LIN {X 0,Y 252.438,Z 584.702,A -85,B 0,C 180,E1 -18965.317,E2 -18965.317} C_VEL
LIN {X 0,Y 250.737,Z 589.425,A -85,B 0,C 180,E1 -18967.666,E2 -18967.666} C_VEL
LIN {X 0,Y 249.329,Z 593.32,A -85,B 0,C 180,E1 -18970.23,E2 -18970.23} C_VEL
LIN {X 0,Y 248.647,Z 595.228,A -85,B 0,C 180,E1 -18971.886,E2 -18971.886} C_VEL
LIN {X 0,Y 247.812,Z 597.412,A -85,B 0,C 180,E1 -18974.635,E2 -18974.635} C_VEL
LIN {X 0,Y 247.334,Z 598.311,A -85,B 0,C 180,E1 -18976.861,E2 -18976.861} C_VEL
LIN {X 0,Y 247.03,Z 598.544,A -85,B 0,C 180,E1 -18978.513,E2 -18978.513} C_VEL
LIN {X 0,Y 246.93,Z 598.348,A -85,B 0,C 180,E1 -18980.168,E2 -18980.168} C_VEL
LIN {X 0,Y 246.961,Z 597.738,A -85,B 0,C 180,E1 -18981.82,E2 -18981.82} C_VEL
LIN {X 0,Y 247.195,Z 596.06,A -85,B 0,C 180,E1 -18984.324,E2 -18984.324} C_VEL
LIN {X 0,Y 247.49,Z 592.461,A -85,B 0,C 180,E1 -18987.559,E2 -18987.559} C_VEL
LIN {X 0,Y 248.083,Z 588.535,A -85,B 0,C 180,E1 -18990,E2 -18990} C_VEL
LIN {X 0,Y 248.817,Z 583.495,A -85,B 0,C 180,E1 -18992.428,E2 -18992.428} C_VEL
LIN {X 0,Y 249.968,Z 577.141,A -85,B 0,C 180,E1 -18994.838,E2 -18994.838} C_VEL
LIN {X 0,Y 251.454,Z 569.206,A -85,B 0,C 180,E1 -18997.225,E2 -18997.225} C_VEL
LIN {X 0,Y 253.19,Z 559.359,A -85,B 0,C 180,E1 -18999.587,E2 -18999.587} C_VEL
LIN {X 0,Y 254.996,Z 549.004,A -85,B 0,C 180,E1 -19001.526,E2 -19001.526} C_VEL
LIN {X 0,Y 256.526,Z 538.775,A -85,B 0,C 180,E1 -19003.063,E2 -19003.063} C_VEL
LIN {X 0,Y 257.87,Z 527.613,A -85,B 0,C 180,E1 -19004.4,E2 -19004.4} C_VEL
LIN {X 0,Y 259.068,Z 516.263,A -85,B 0,C 180,E1 -19005.438,E2 -19005.438} C_VEL
LIN {X 0,Y 260.042,Z 503.315,A -85,B 0,C 180,E1 -19006.284,E2 -19006.284} C_VEL
LIN {X 0,Y 260.587,Z 491.019,A -85,B 0,C 180,E1 -19006.803,E2 -19006.803} C_VEL
LIN {X 0,Y 262.544,Z 423.316,A -85,B 0,C 180,E1 -19008.621,E2 -19008.621} C_VEL
LIN {X 0,Y 256.099,Z 405.689,A -85,B 0,C 180,E1 -19009.811,E2 -19009.811} C_VEL
LIN {X 0,Y 249.864,Z 392.807,A -85,B 0,C 180,E1 -19010.9,E2 -19010.9} C_VEL
LIN {X 0,Y 249.121,Z 390.454,A -85,B 0,C 180,E1 -19011.108,E2 -19011.108} C_VEL
LIN {X 0,Y 249.136,Z 390.441,A -85,B 0,C 180,E1 -19015.482,E2 -19015.482} C_VEL
LIN {X 0,Y 249.09,Z 390.455,A -85,B 0,C 180,E1 -19018.994,E2 -19018.994} C_VEL
LIN {X 0,Y 249.035,Z 390.465,A -85,B 0,C 180,E1 -19022.424,E2 -19022.424} C_VEL
LIN {X 0,Y 249.059,Z 390.462,A -85,B 0,C 180,E1 -19026.339,E2 -19026.339} C_VEL
LIN {X 0,Y 249.008,Z 390.46,A -85,B 0,C 180,E1 -19030.477,E2 -19030.477} C_VEL
LIN {X 0,Y 249.018,Z 390.463,A -85,B 0,C 180,E1 -19034.874,E2 -19034.874} C_VEL
LIN {X 0,Y 249.08,Z 390.445,A -85,B 0,C 180,E1 -19037.376,E2 -19037.376} C_VEL
LIN {X 0,Y 249.052,Z 390.46,A -85,B 0,C 180,E1 -19041.623,E2 -19041.623} C_VEL
LIN {X 0,Y 249.059,Z 390.445,A -85,B 0,C 180,E1 -19045.641,E2 -19045.641} C_VEL
LIN {X 0,Y 249.045,Z 390.461,A -85,B 0,C 180,E1 -19049.471,E2 -19049.471} C_VEL
LIN {X 0,Y 249.068,Z 390.449,A -85,B 0,C 180,E1 -19053.161,E2 -19053.161} C_VEL
LIN {X 0,Y 249.081,Z 390.455,A -85,B 0,C 180,E1 -19056.732,E2 -19056.732} C_VEL
LIN {X 0,Y 249.127,Z 390.453,A -85,B 0,C 180,E1 -19060.212,E2 -19060.212} C_VEL
LIN {X 0,Y 249.238,Z 390.426,A -85,B 0,C 180,E1 -19063.621,E2 -19063.621} C_VEL
LIN {X 0,Y 249.248,Z 390.436,A -85,B 0,C 180,E1 -19068.616,E2 -19068.616} C_VEL
LIN {X 0,Y 249.476,Z 390.406,A -85,B 0,C 180,E1 -19071.902,E2 -19071.902} C_VEL
LIN {X 0,Y 249.431,Z 390.406,A -85,B 0,C 180,E1 -19076.769,E2 -19076.769} C_VEL
LIN {X 0,Y 249.73,Z 390.378,A -85,B 0,C 180,E1 -19080,E2 -19080} C_VEL
LIN {X 0,Y 249.432,Z 390.408,A -85,B 0,C 180,E1 -19083.23,E2 -19083.23} C_VEL
LIN {X 0,Y 249.476,Z 390.407,A -85,B 0,C 180,E1 -19088.097,E2 -19088.097} C_VEL
LIN {X 0,Y 249.354,Z 390.421,A -85,B 0,C 180,E1 -19089.954,E2 -19089.954} C_VEL
LIN {X 0,Y 248.581,Z 390.52,A -85,B 0,C 180,E1 -19091.3,E2 -19091.3} C_VEL
LIN {X 0,Y 245.714,Z 390.878,A -85,B 0,C 180,E1 -19093.495,E2 -19093.495} C_VEL
LIN {X 0,Y 242.486,Z 391.281,A -85,B 0,C 180,E1 -19096.2,E2 -19096.2} C_VEL
LIN {X 0,Y 242.121,Z 391.321,A -85,B 0,C 180,E1 -19097.136,E2 -19097.136} C_VEL
LIN {X 0,Y 242.045,Z 391.335,A -85,B 0,C 180,E1 -19102.177,E2 -19102.177} C_VEL
LIN {X 0,Y 242.062,Z 391.335,A -85,B 0,C 180,E1 -19105.838,E2 -19105.838} C_VEL
LIN {X 0,Y 242.003,Z 391.34,A -85,B 0,C 180,E1 -19109.584,E2 -19109.584} C_VEL
LIN {X 0,Y 241.987,Z 391.343,A -85,B 0,C 180,E1 -19113.491,E2 -19113.491} C_VEL
LIN {X 0,Y 242.009,Z 391.34,A -85,B 0,C 180,E1 -19117.578,E2 -19117.578} C_VEL
LIN {X 0,Y 241.982,Z 391.342,A -85,B 0,C 180,E1 -19121.913,E2 -19121.913} C_VEL
LIN {X 0,Y 241.97,Z 391.344,A -85,B 0,C 180,E1 -19126.562,E2 -19126.562} C_VEL
LIN {X 0,Y 241.976,Z 391.346,A -85,B 0,C 180,E1 -19130.286,E2 -19130.286} C_VEL
LIN {X 0,Y 242.073,Z 391.536,A -85,B 0,C 180,E1 -19132.906,E2 -19132.906} C_VEL
LIN {X 0,Y 244.318,Z 401.427,A -85,B 0,C 180,E1 -19136.87,E2 -19136.87} C_VEL
LIN {X 0,Y 245.764,Z 408.526,A -85,B 0,C 180,E1 -19139.488,E2 -19139.488} C_VEL
LIN {X 0,Y 250.251,Z 420.691,A -85,B 0,C 180,E1 -19140.38,E2 -19140.38} C_VEL
LIN {X 0,Y 254.146,Z 451.891,A -85,B 0,C 180,E1 -19141.755,E2 -19141.755} C_VEL
LIN {X 0,Y 255.201,Z 463.108,A -85,B 0,C 180,E1 -19142.202,E2 -19142.202} C_VEL
LIN {X 0,Y 253.446,Z 517.374,A -85,B 0,C 180,E1 -19143.717,E2 -19143.717} C_VEL
LIN {X 0,Y 252.497,Z 530.59,A -85,B 0,C 180,E1 -19144.387,E2 -19144.387} C_VEL
LIN {X 0,Y 251.165,Z 542.728,A -85,B 0,C 180,E1 -19145.294,E2 -19145.294} C_VEL
LIN {X 0,Y 249.537,Z 554.986,A -85,B 0,C 180,E1 -19146.559,E2 -19146.559} C_VEL
LIN {X 0,Y 247.702,Z 566.611,A -85,B 0,C 180,E1 -19148.137,E2 -19148.137} C_VEL
LIN {X 0,Y 245.775,Z 577.065,A -85,B 0,C 180,E1 -19149.932,E2 -19149.932} C_VEL
LIN {X 0,Y 244.06,Z 587.411,A -85,B 0,C 180,E1 -19152.213,E2 -19152.213} C_VEL
LIN {X 0,Y 242.628,Z 595.579,A -85,B 0,C 180,E1 -19154.459,E2 -19154.459} C_VEL
LIN {X 0,Y 241.355,Z 602.896,A -85,B 0,C 180,E1 -19156.958,E2 -19156.958} C_VEL
LIN {X 0,Y 240.678,Z 607.838,A -85,B 0,C 180,E1 -19159.059,E2 -19159.059} C_VEL
LIN {X 0,Y 240.168,Z 612.631,A -85,B 0,C 180,E1 -19161.587,E2 -19161.587} C_VEL
LIN {X 0,Y 239.979,Z 615.204,A -85,B 0,C 180,E1 -19163.273,E2 -19163.273} C_VEL
LIN {X 0,Y 239.92,Z 617.267,A -85,B 0,C 180,E1 -19164.958,E2 -19164.958} C_VEL
LIN {X 0,Y 239.952,Z 618.906,A -85,B 0,C 180,E1 -19166.642,E2 -19166.642} C_VEL
LIN {X 0,Y 240.006,Z 620.132,A -85,B 0,C 180,E1 -19168.322,E2 -19168.322} C_VEL
LIN {X 0,Y 240.02,Z 620.919,A -85,B 0,C 180,E1 -19170,E2 -19170} C_VEL
LIN {X 0,Y 239.975,Z 621.281,A -85,B 0,C 180,E1 -19171.678,E2 -19171.678} C_VEL
LIN {X 0,Y 239.902,Z 621.251,A -85,B 0,C 180,E1 -19173.359,E2 -19173.359} C_VEL
LIN {X 0,Y 239.845,Z 620.834,A -85,B 0,C 180,E1 -19175.043,E2 -19175.043} C_VEL
LIN {X 0,Y 239.9,Z 620.017,A -85,B 0,C 180,E1 -19176.729,E2 -19176.729} C_VEL
LIN {X 0,Y 240.552,Z 617.129,A -85,B 0,C 180,E1 -19180.096,E2 -19180.096} C_VEL
LIN {X 0,Y 241.429,Z 613.857,A -85,B 0,C 180,E1 -19182.61,E2 -19182.61} C_VEL
LIN {X 0,Y 242.806,Z 609.541,A -85,B 0,C 180,E1 -19185.1,E2 -19185.1} C_VEL
LIN {X 0,Y 244.64,Z 604.063,A -85,B 0,C 180,E1 -19187.556,E2 -19187.556} C_VEL
LIN {X 0,Y 246.842,Z 597.119,A -85,B 0,C 180,E1 -19190.021,E2 -19190.021} C_VEL
LIN {X 0,Y 249.439,Z 588.791,A -85,B 0,C 180,E1 -19192.356,E2 -19192.356} C_VEL
LIN {X 0,Y 252.13,Z 580.114,A -85,B 0,C 180,E1 -19194.276,E2 -19194.276} C_VEL
LIN {X 0,Y 255.107,Z 569.459,A -85,B 0,C 180,E1 -19196.153,E2 -19196.153} C_VEL
LIN {X 0,Y 257.715,Z 558.887,A -85,B 0,C 180,E1 -19197.619,E2 -19197.619} C_VEL
LIN {X 0,Y 260.14,Z 547.118,A -85,B 0,C 180,E1 -19198.875,E2 -19198.875} C_VEL
LIN {X 0,Y 262.356,Z 533.614,A -85,B 0,C 180,E1 -19199.928,E2 -19199.928} C_VEL
LIN {X 0,Y 263.864,Z 520.48,A -85,B 0,C 180,E1 -19200.622,E2 -19200.622} C_VEL
LIN {X 0,Y 264.804,Z 504.801,A -85,B 0,C 180,E1 -19201.107,E2 -19201.107} C_VEL
LIN {X 0,Y 266.35,Z 464.818,A -85,B 0,C 180,E1 -19202.171,E2 -19202.171} C_VEL
LIN {X 0,Y 262.808,Z 441.78,A -85,B 0,C 180,E1 -19203.496,E2 -19203.496} C_VEL
LIN {X 0,Y 261.785,Z 438.425,A -85,B 0,C 180,E1 -19203.778,E2 -19203.778} C_VEL
LIN {X 0,Y 254.825,Z 423.393,A -85,B 0,C 180,E1 -19205.508,E2 -19205.508} C_VEL
LIN {X 0,Y 248.373,Z 411.073,A -85,B 0,C 180,E1 -19207.183,E2 -19207.183} C_VEL
LIN {X 0,Y 246.244,Z 406.811,A -85,B 0,C 180,E1 -19207.795,E2 -19207.795} C_VEL
LIN {X 0,Y 243.975,Z 398.341,A -85,B 0,C 180,E1 -19211.889,E2 -19211.889} C_VEL
LIN {X 0,Y 241.967,Z 391.337,A -85,B 0,C 180,E1 -19215.683,E2 -19215.683} C_VEL
LIN {X 0,Y 242.005,Z 391.335,A -85,B 0,C 180,E1 -19220.291,E2 -19220.291} C_VEL
LIN {X 0,Y 242.033,Z 391.333,A -85,B 0,C 180,E1 -19224.497,E2 -19224.497} C_VEL
LIN {X 0,Y 241.972,Z 391.344,A -85,B 0,C 180,E1 -19228.48,E2 -19228.48} C_VEL
LIN {X 0,Y 242.005,Z 391.336,A -85,B 0,C 180,E1 -19232.313,E2 -19232.313} C_VEL
LIN {X 0,Y 242.052,Z 391.304,A -85,B 0,C 180,E1 -19236.016,E2 -19236.016} C_VEL
LIN {X 0,Y 242.032,Z 391.333,A -85,B 0,C 180,E1 -19239.608,E2 -19239.608} C_VEL
LIN {X 0,Y 242.159,Z 391.32,A -85,B 0,C 180,E1 -19243.278,E2 -19243.278} C_VEL
LIN {X 0,Y 242.181,Z 391.314,A -85,B 0,C 180,E1 -19248.28,E2 -19248.28} C_VEL
LIN {X 0,Y 242.422,Z 391.288,A -85,B 0,C 180,E1 -19251.666,E2 -19251.666} C_VEL
LIN {X 0,Y 242.256,Z 391.3,A -85,B 0,C 180,E1 -19255.008,E2 -19255.008} C_VEL
LIN {X 0,Y 242.632,Z 391.252,A -85,B 0,C 180,E1 -19258.341,E2 -19258.341} C_VEL
LIN {X 0,Y 242.632,Z 391.261,A -85,B 0,C 180,E1 -19261.66,E2 -19261.66} C_VEL
LIN {X 0,Y 242.416,Z 391.285,A -85,B 0,C 180,E1 -19266.7,E2 -19266.7} C_VEL
LIN {X 0,Y 242.263,Z 391.307,A -85,B 0,C 180,E1 -19270.024,E2 -19270.024} C_VEL
LIN {X 0,Y 242.152,Z 391.321,A -85,B 0,C 180,E1 -19275.142,E2 -19275.142} C_VEL
LIN {X 0,Y 242.067,Z 391.332,A -85,B 0,C 180,E1 -19278.625,E2 -19278.625} C_VEL
LIN {X 0,Y 242.01,Z 391.336,A -85,B 0,C 180,E1 -19282.181,E2 -19282.181} C_VEL
LIN {X 0,Y 242.064,Z 391.303,A -85,B 0,C 180,E1 -19285.839,E2 -19285.839} C_VEL
LIN {X 0,Y 242.028,Z 391.337,A -85,B 0,C 180,E1 -19289.581,E2 -19289.581} C_VEL
LIN {X 0,Y 241.989,Z 391.34,A -85,B 0,C 180,E1 -19293.492,E2 -19293.492} C_VEL
LIN {X 0,Y 242.012,Z 391.34,A -85,B 0,C 180,E1 -19297.579,E2 -19297.579} C_VEL
LIN {X 0,Y 242.011,Z 391.33,A -85,B 0,C 180,E1 -19302.257,E2 -19302.257} C_VEL
LIN {X 0,Y 242.037,Z 391.38,A -85,B 0,C 180,E1 -19302.426,E2 -19302.426} C_VEL
LIN {X 0,Y 243,Z 394.117,A -85,B 0,C 180,E1 -19302.743,E2 -19302.743} C_VEL
LIN {X 0,Y 244.946,Z 396.585,A -85,B 0,C 180,E1 -19303.254,E2 -19303.254} C_VEL
LIN {X 0,Y 247.23,Z 400.091,A -85,B 0,C 180,E1 -19303.862,E2 -19303.862} C_VEL
LIN {X 0,Y 255.012,Z 412.382,A -85,B 0,C 180,E1 -19305.821,E2 -19305.821} C_VEL
LIN {X 0,Y 263.08,Z 428.015,A -85,B 0,C 180,E1 -19307.774,E2 -19307.774} C_VEL
LIN {X 0,Y 267.366,Z 437.539,A -85,B 0,C 180,E1 -19308.784,E2 -19308.784} C_VEL
LIN {X 0,Y 264.97,Z 495.594,A -85,B 0,C 180,E1 -19310.35,E2 -19310.35} C_VEL
LIN {X 0,Y 263.881,Z 508.231,A -85,B 0,C 180,E1 -19310.948,E2 -19310.948} C_VEL
LIN {X 0,Y 262.362,Z 520.8,A -85,B 0,C 180,E1 -19311.847,E2 -19311.847} C_VEL
LIN {X 0,Y 260.022,Z 533.292,A -85,B 0,C 180,E1 -19313.032,E2 -19313.032} C_VEL
LIN {X 0,Y 257.962,Z 543.738,A -85,B 0,C 180,E1 -19314.385,E2 -19314.385} C_VEL
LIN {X 0,Y 255.307,Z 554.907,A -85,B 0,C 180,E1 -19316.213,E2 -19316.213} C_VEL
LIN {X 0,Y 252.658,Z 564.11,A -85,B 0,C 180,E1 -19318.096,E2 -19318.096} C_VEL
LIN {X 0,Y 249.896,Z 573.004,A -85,B 0,C 180,E1 -19320.417,E2 -19320.417} C_VEL
LIN {X 0,Y 247.328,Z 580.664,A -85,B 0,C 180,E1 -19322.958,E2 -19322.958} C_VEL
LIN {X 0,Y 245.192,Z 586.513,A -85,B 0,C 180,E1 -19325.442,E2 -19325.442} C_VEL
LIN {X 0,Y 243.424,Z 591.073,A -85,B 0,C 180,E1 -19327.956,E2 -19327.956} C_VEL
LIN {X 0,Y 242.515,Z 593.457,A -85,B 0,C 180,E1 -19329.65,E2 -19329.65} C_VEL
LIN {X 0,Y 241.743,Z 595.398,A -85,B 0,C 180,E1 -19331.35,E2 -19331.35} C_VEL
LIN {X 0,Y 240.777,Z 597.793,A -85,B 0,C 180,E1 -19334.417,E2 -19334.417} C_VEL
LIN {X 0,Y 240.304,Z 598.604,A -85,B 0,C 180,E1 -19336.469,E2 -19336.469} C_VEL
LIN {X 0,Y 239.984,Z 598.866,A -85,B 0,C 180,E1 -19338.171,E2 -19338.171} C_VEL
LIN {X 0,Y 239.854,Z 598.727,A -85,B 0,C 180,E1 -19339.875,E2 -19339.875} C_VEL
LIN {X 0,Y 239.855,Z 598.151,A -85,B 0,C 180,E1 -19341.576,E2 -19341.576} C_VEL
LIN {X 0,Y 240.104,Z 596.325,A -85,B 0,C 180,E1 -19344.394,E2 -19344.394} C_VEL
LIN {X 0,Y 240.395,Z 592.995,A -85,B 0,C 180,E1 -19347.487,E2 -19347.487} C_VEL
LIN {X 0,Y 241.006,Z 589.135,A -85,B 0,C 180,E1 -19350,E2 -19350} C_VEL
LIN {X 0,Y 241.75,Z 584.167,A -85,B 0,C 180,E1 -19352.499,E2 -19352.499} C_VEL
LIN {X 0,Y 242.919,Z 577.919,A -85,B 0,C 180,E1 -19354.979,E2 -19354.979} C_VEL
LIN {X 0,Y 244.449,Z 570.093,A -85,B 0,C 180,E1 -19357.433,E2 -19357.433} C_VEL
LIN {X 0,Y 246.24,Z 560.358,A -85,B 0,C 180,E1 -19359.86,E2 -19359.86} C_VEL
LIN {X 0,Y 248.079,Z 550.21,A -85,B 0,C 180,E1 -19361.852,E2 -19361.852} C_VEL
LIN {X 0,Y 249.88,Z 538.746,A -85,B 0,C 180,E1 -19363.624,E2 -19363.624} C_VEL
LIN {X 0,Y 251.274,Z 527.501,A -85,B 0,C 180,E1 -19364.994,E2 -19364.994} C_VEL
LIN {X 0,Y 252.521,Z 515.971,A -85,B 0,C 180,E1 -19366.055,E2 -19366.055} C_VEL
LIN {X 0,Y 253.531,Z 502.731,A -85,B 0,C 180,E1 -19366.921,E2 -19366.921} C_VEL
LIN {X 0,Y 254.11,Z 489.846,A -85,B 0,C 180,E1 -19367.452,E2 -19367.452} C_VEL
LIN {X 0,Y 256.075,Z 424.887,A -85,B 0,C 180,E1 -19369.228,E2 -19369.228} C_VEL
LIN {X 0,Y 249.533,Z 407.216,A -85,B 0,C 180,E1 -19370.483,E2 -19370.483} C_VEL
LIN {X 0,Y 243.117,Z 394.259,A -85,B 0,C 180,E1 -19371.647,E2 -19371.647} C_VEL
LIN {X 0,Y 242.108,Z 391.841,A -85,B 0,C 180,E1 -19371.849,E2 -19371.849} C_VEL
LIN {X 0,Y 242.037,Z 391.338,A -85,B 0,C 180,E1 -19371.924,E2 -19371.924} C_VEL
LIN {X 0,Y 242.069,Z 391.322,A -85,B 0,C 180,E1 -19375.837,E2 -19375.837} C_VEL
LIN {X 0,Y 242.034,Z 391.333,A -85,B 0,C 180,E1 -19379.579,E2 -19379.579} C_VEL
LIN {X 0,Y 241.989,Z 391.341,A -85,B 0,C 180,E1 -19383.49,E2 -19383.49} C_VEL
LIN {X 0,Y 241.992,Z 391.339,A -85,B 0,C 180,E1 -19387.58,E2 -19387.58} C_VEL
LIN {X 0,Y 241.943,Z 391.339,A -85,B 0,C 180,E1 -19391.92,E2 -19391.92} C_VEL
LIN {X 0,Y 242.001,Z 391.329,A -85,B 0,C 180,E1 -19396.553,E2 -19396.553} C_VEL
LIN {X 0,Y 242.01,Z 391.338,A -85,B 0,C 180,E1 -19400.291,E2 -19400.291} C_VEL
LIN {X 0,Y 242.035,Z 391.322,A -85,B 0,C 180,E1 -19404.496,E2 -19404.496} C_VEL
LIN {X 0,Y 241.972,Z 391.344,A -85,B 0,C 180,E1 -19408.479,E2 -19408.479} C_VEL
LIN {X 0,Y 241.999,Z 391.333,A -85,B 0,C 180,E1 -19412.311,E2 -19412.311} C_VEL
LIN {X 0,Y 242.057,Z 391.323,A -85,B 0,C 180,E1 -19416.015,E2 -19416.015} C_VEL
LIN {X 0,Y 242.057,Z 391.332,A -85,B 0,C 180,E1 -19419.609,E2 -19419.609} C_VEL
LIN {X 0,Y 242.16,Z 391.308,A -85,B 0,C 180,E1 -19423.277,E2 -19423.277} C_VEL
LIN {X 0,Y 242.182,Z 391.317,A -85,B 0,C 180,E1 -19428.279,E2 -19428.279} C_VEL
LIN {X 0,Y 242.423,Z 391.285,A -85,B 0,C 180,E1 -19431.665,E2 -19431.665} C_VEL
LIN {X 0,Y 242.254,Z 391.287,A -85,B 0,C 180,E1 -19435.007,E2 -19435.007} C_VEL
LIN {X 0,Y 242.632,Z 391.259,A -85,B 0,C 180,E1 -19438.34,E2 -19438.34} C_VEL
LIN {X 0,Y 242.632,Z 391.261,A -85,B 0,C 180,E1 -19441.659,E2 -19441.659} C_VEL
LIN {X 0,Y 242.428,Z 391.285,A -85,B 0,C 180,E1 -19446.659,E2 -19446.659} C_VEL
LIN {X 0,Y 242.309,Z 391.301,A -85,B 0,C 180,E1 -19450.022,E2 -19450.022} C_VEL
LIN {X 0,Y 242.159,Z 391.318,A -85,B 0,C 180,E1 -19455.141,E2 -19455.141} C_VEL
LIN {X 0,Y 242.121,Z 391.321,A -85,B 0,C 180,E1 -19457.136,E2 -19457.136} C_VEL
LIN {X 0,Y 241.359,Z 391.416,A -85,B 0,C 180,E1 -19458.525,E2 -19458.525} C_VEL
LIN {X 0,Y 238.423,Z 391.785,A -85,B 0,C 180,E1 -19460.789,E2 -19460.789} C_VEL
LIN {X 0,Y 236.011,Z 392.084,A -85,B 0,C 180,E1 -19462.634,E2 -19462.634} C_VEL
LIN {X 0,Y 235.027,Z 392.207,A -85,B 0,C 180,E1 -19464.067,E2 -19464.067} C_VEL
LIN {X 0,Y 234.971,Z 392.213,A -85,B 0,C 180,E1 -19464.552,E2 -19464.552} C_VEL
LIN {X 0,Y 234.933,Z 392.22,A -85,B 0,C 180,E1 -19468.596,E2 -19468.596} C_VEL
LIN {X 0,Y 234.946,Z 392.219,A -85,B 0,C 180,E1 -19473.117,E2 -19473.117} C_VEL
LIN {X 0,Y 234.943,Z 392.219,A -85,B 0,C 180,E1 -19476.746,E2 -19476.746} C_VEL
LIN {X 0,Y 234.942,Z 392.219,A -85,B 0,C 180,E1 -19481.155,E2 -19481.155} C_VEL
LIN {X 0,Y 234.937,Z 392.22,A -85,B 0,C 180,E1 -19484.116,E2 -19484.116} C_VEL
LIN {X 0,Y 234.926,Z 392.224,A -85,B 0,C 180,E1 -19488.408,E2 -19488.408} C_VEL
LIN {X 0,Y 234.991,Z 392.246,A -85,B 0,C 180,E1 -19492.187,E2 -19492.187} C_VEL
LIN {X 0,Y 237.125,Z 401.604,A -85,B 0,C 180,E1 -19496.086,E2 -19496.086} C_VEL
LIN {X 0,Y 238.403,Z 407.841,A -85,B 0,C 180,E1 -19498.557,E2 -19498.557} C_VEL
LIN {X 0,Y 244.062,Z 422.946,A -85,B 0,C 180,E1 -19499.755,E2 -19499.755} C_VEL
LIN {X 0,Y 247.913,Z 455.05,A -85,B 0,C 180,E1 -19501.204,E2 -19501.204} C_VEL
LIN {X 0,Y 248.73,Z 462.941,A -85,B 0,C 180,E1 -19501.537,E2 -19501.537} C_VEL
LIN {X 0,Y 246.886,Z 516.957,A -85,B 0,C 180,E1 -19503.077,E2 -19503.077} C_VEL
LIN {X 0,Y 245.941,Z 530.212,A -85,B 0,C 180,E1 -19503.767,E2 -19503.767} C_VEL
LIN {X 0,Y 244.574,Z 542.364,A -85,B 0,C 180,E1 -19504.695,E2 -19504.695} C_VEL
LIN {X 0,Y 243.04,Z 553.832,A -85,B 0,C 180,E1 -19505.893,E2 -19505.893} C_VEL
LIN {X 0,Y 241.057,Z 565.602,A -85,B 0,C 180,E1 -19507.502,E2 -19507.502} C_VEL
LIN {X 0,Y 239.084,Z 576.176,A -85,B 0,C 180,E1 -19509.345,E2 -19509.345} C_VEL
LIN {X 0,Y 237.224,Z 586.425,A -85,B 0,C 180,E1 -19511.623,E2 -19511.623} C_VEL
LIN {X 0,Y 236.313,Z 592.065,A -85,B 0,C 180,E1 -19513.144,E2 -19513.144} C_VEL
LIN {X 0,Y 234.865,Z 600.014,A -85,B 0,C 180,E1 -19515.708,E2 -19515.708} C_VEL
LIN {X 0,Y 233.893,Z 605.396,A -85,B 0,C 180,E1 -19517.858,E2 -19517.858} C_VEL
LIN {X 0,Y 233.263,Z 610.656,A -85,B 0,C 180,E1 -19520.462,E2 -19520.462} C_VEL
LIN {X 0,Y 232.902,Z 614.724,A -85,B 0,C 180,E1 -19523.067,E2 -19523.067} C_VEL
LIN {X 0,Y 232.84,Z 616.933,A -85,B 0,C 180,E1 -19524.914,E2 -19524.914} C_VEL
LIN {X 0,Y 232.934,Z 619.728,A -85,B 0,C 180,E1 -19528.271,E2 -19528.271} C_VEL
LIN {X 0,Y 232.948,Z 620.554,A -85,B 0,C 180,E1 -19530,E2 -19530} C_VEL
LIN {X 0,Y 232.903,Z 620.937,A -85,B 0,C 180,E1 -19531.729,E2 -19531.729} C_VEL
LIN {X 0,Y 232.747,Z 620.643,A -85,B 0,C 180,E1 -19534.821,E2 -19534.821} C_VEL
LIN {X 0,Y 232.821,Z 619.746,A -85,B 0,C 180,E1 -19536.935,E2 -19536.935} C_VEL
LIN {X 0,Y 233.11,Z 618.53,A -85,B 0,C 180,E1 -19538.67,E2 -19538.67} C_VEL
LIN {X 0,Y 234.134,Z 614.877,A -85,B 0,C 180,E1 -19542.129,E2 -19542.129} C_VEL
LIN {X 0,Y 235.377,Z 610.962,A -85,B 0,C 180,E1 -19544.702,E2 -19544.702} C_VEL
LIN {X 0,Y 237.202,Z 605.943,A -85,B 0,C 180,E1 -19547.234,E2 -19547.234} C_VEL
LIN {X 0,Y 239.6,Z 598.918,A -85,B 0,C 180,E1 -19549.994,E2 -19549.994} C_VEL
LIN {X 0,Y 242.371,Z 590.36,A -85,B 0,C 180,E1 -19552.594,E2 -19552.594} C_VEL
LIN {X 0,Y 245.076,Z 582.116,A -85,B 0,C 180,E1 -19554.57,E2 -19554.57} C_VEL
LIN {X 0,Y 248.107,Z 572.065,A -85,B 0,C 180,E1 -19556.496,E2 -19556.496} C_VEL
LIN {X 0,Y 250.761,Z 562.126,A -85,B 0,C 180,E1 -19557.998,E2 -19557.998} C_VEL
LIN {X 0,Y 253.206,Z 551.351,A -85,B 0,C 180,E1 -19559.287,E2 -19559.287} C_VEL
LIN {X 0,Y 255.688,Z 538.366,A -85,B 0,C 180,E1 -19560.449,E2 -19560.449} C_VEL
LIN {X 0,Y 257.456,Z 525.828,A -85,B 0,C 180,E1 -19561.242,E2 -19561.242} C_VEL
LIN {X 0,Y 258.612,Z 513.139,A -85,B 0,C 180,E1 -19561.756,E2 -19561.756} C_VEL
LIN {X 0,Y 260.622,Z 466.258,A -85,B 0,C 180,E1 -19563.028,E2 -19563.028} C_VEL
LIN {X 0,Y 257.252,Z 443.764,A -85,B 0,C 180,E1 -19564.362,E2 -19564.362} C_VEL
LIN {X 0,Y 253.327,Z 434.502,A -85,B 0,C 180,E1 -19565.385,E2 -19565.385} C_VEL
LIN {X 0,Y 246.597,Z 420.628,A -85,B 0,C 180,E1 -19567.177,E2 -19567.177} C_VEL
LIN {X 0,Y 241.116,Z 410.641,A -85,B 0,C 180,E1 -19568.7,E2 -19568.7} C_VEL
LIN {X 0,Y 238.83,Z 406.306,A -85,B 0,C 180,E1 -19569.419,E2 -19569.419} C_VEL
LIN {X 0,Y 236.687,Z 398.366,A -85,B 0,C 180,E1 -19573.494,E2 -19573.494} C_VEL
LIN {X 0,Y 234.929,Z 392.214,A -85,B 0,C 180,E1 -19577.035,E2 -19577.035} C_VEL
LIN {X 0,Y 234.952,Z 392.213,A -85,B 0,C 180,E1 -19581.086,E2 -19581.086} C_VEL
LIN {X 0,Y 234.957,Z 392.216,A -85,B 0,C 180,E1 -19585.367,E2 -19585.367} C_VEL
LIN {X 0,Y 234.965,Z 392.211,A -85,B 0,C 180,E1 -19590.157,E2 -19590.157} C_VEL
LIN {X 0,Y 234.99,Z 392.186,A -85,B 0,C 180,E1 -19593.793,E2 -19593.793} C_VEL
LIN {X 0,Y 235.007,Z 392.213,A -85,B 0,C 180,E1 -19598.97,E2 -19598.97} C_VEL
LIN {X 0,Y 235.092,Z 392.202,A -85,B 0,C 180,E1 -19603.059,E2 -19603.059} C_VEL
LIN {X 0,Y 235.141,Z 392.193,A -85,B 0,C 180,E1 -19607.924,E2 -19607.924} C_VEL
LIN {X 0,Y 235.372,Z 392.167,A -85,B 0,C 180,E1 -19611.414,E2 -19611.414} C_VEL
LIN {X 0,Y 235.399,Z 392.155,A -85,B 0,C 180,E1 -19613.142,E2 -19613.142} C_VEL
LIN {X 0,Y 235.591,Z 392.129,A -85,B 0,C 180,E1 -19618.291,E2 -19618.291} C_VEL
LIN {X 0,Y 235.591,Z 392.138,A -85,B 0,C 180,E1 -19621.71,E2 -19621.71} C_VEL
LIN {X 0,Y 235.369,Z 392.162,A -85,B 0,C 180,E1 -19626.86,E2 -19626.86} C_VEL
LIN {X 0,Y 235.21,Z 392.187,A -85,B 0,C 180,E1 -19630.328,E2 -19630.328} C_VEL
LIN {X 0,Y 235.103,Z 392.198,A -85,B 0,C 180,E1 -19635.608,E2 -19635.608} C_VEL
LIN {X 0,Y 235.004,Z 392.212,A -85,B 0,C 180,E1 -19639.207,E2 -19639.207} C_VEL
LIN {X 0,Y 234.958,Z 392.219,A -85,B 0,C 180,E1 -19642.884,E2 -19642.884} C_VEL
LIN {X 0,Y 234.967,Z 392.185,A -85,B 0,C 180,E1 -19646.658,E2 -19646.658} C_VEL
LIN {X 0,Y 234.93,Z 392.217,A -85,B 0,C 180,E1 -19650.569,E2 -19650.569} C_VEL
LIN {X 0,Y 234.959,Z 392.215,A -85,B 0,C 180,E1 -19654.634,E2 -19654.634} C_VEL
LIN {X 0,Y 234.966,Z 392.217,A -85,B 0,C 180,E1 -19658.953,E2 -19658.953} C_VEL
LIN {X 0,Y 235.004,Z 392.395,A -85,B 0,C 180,E1 -19660.859,E2 -19660.859} C_VEL
LIN {X 0,Y 235.907,Z 394.961,A -85,B 0,C 180,E1 -19661.18,E2 -19661.18} C_VEL
LIN {X 0,Y 238.169,Z 397.681,A -85,B 0,C 180,E1 -19661.815,E2 -19661.815} C_VEL
LIN {X 0,Y 240.353,Z 401.021,A -85,B 0,C 180,E1 -19662.44,E2 -19662.44} C_VEL
LIN {X 0,Y 249.114,Z 414.608,A -85,B 0,C 180,E1 -19664.784,E2 -19664.784} C_VEL
LIN {X 0,Y 255.056,Z 425.681,A -85,B 0,C 180,E1 -19666.303,E2 -19666.303} C_VEL
LIN {X 0,Y 261.654,Z 439.842,A -85,B 0,C 180,E1 -19667.937,E2 -19667.937} C_VEL
LIN {X 0,Y 259.126,Z 496.783,A -85,B 0,C 180,E1 -19669.505,E2 -19669.505} C_VEL
LIN {X 0,Y 257.971,Z 509.205,A -85,B 0,C 180,E1 -19670.115,E2 -19670.115} C_VEL
LIN {X 0,Y 256.351,Z 521.736,A -85,B 0,C 180,E1 -19671.036,E2 -19671.036} C_VEL
LIN {X 0,Y 253.924,Z 534.044,A -85,B 0,C 180,E1 -19672.24,E2 -19672.24} C_VEL
LIN {X 0,Y 251.772,Z 544.409,A -85,B 0,C 180,E1 -19673.618,E2 -19673.618} C_VEL
LIN {X 0,Y 249.241,Z 554.678,A -85,B 0,C 180,E1 -19675.331,E2 -19675.331} C_VEL
LIN {X 0,Y 246.521,Z 563.78,A -85,B 0,C 180,E1 -19677.204,E2 -19677.204} C_VEL
LIN {X 0,Y 243.912,Z 571.884,A -85,B 0,C 180,E1 -19679.289,E2 -19679.289} C_VEL
LIN {X 0,Y 241.314,Z 579.451,A -85,B 0,C 180,E1 -19681.754,E2 -19681.754} C_VEL
LIN {X 0,Y 238.603,Z 586.513,A -85,B 0,C 180,E1 -19684.717,E2 -19684.717} C_VEL
LIN {X 0,Y 236.709,Z 591.157,A -85,B 0,C 180,E1 -19687.296,E2 -19687.296} C_VEL
LIN {X 0,Y 235.725,Z 593.593,A -85,B 0,C 180,E1 -19689.037,E2 -19689.037} C_VEL
LIN {X 0,Y 234.88,Z 595.567,A -85,B 0,C 180,E1 -19690.784,E2 -19690.784} C_VEL
LIN {X 0,Y 234.227,Z 597.116,A -85,B 0,C 180,E1 -19692.54,E2 -19692.54} C_VEL
LIN {X 0,Y 233.709,Z 598.22,A -85,B 0,C 180,E1 -19694.298,E2 -19694.298} C_VEL
LIN {X 0,Y 233.286,Z 598.897,A -85,B 0,C 180,E1 -19696.054,E2 -19696.054} C_VEL
LIN {X 0,Y 232.796,Z 599.09,A -85,B 0,C 180,E1 -19699.564,E2 -19699.564} C_VEL
LIN {X 0,Y 232.772,Z 598.563,A -85,B 0,C 180,E1 -19701.317,E2 -19701.317} C_VEL
LIN {X 0,Y 233.032,Z 596.63,A -85,B 0,C 180,E1 -19704.419,E2 -19704.419} C_VEL
LIN {X 0,Y 233.303,Z 593.527,A -85,B 0,C 180,E1 -19707.41,E2 -19707.41} C_VEL
LIN {X 0,Y 233.929,Z 589.732,A -85,B 0,C 180,E1 -19710,E2 -19710} C_VEL
LIN {X 0,Y 234.685,Z 584.835,A -85,B 0,C 180,E1 -19712.575,E2 -19712.575} C_VEL
LIN {X 0,Y 235.871,Z 578.669,A -85,B 0,C 180,E1 -19715.128,E2 -19715.128} C_VEL
LIN {X 0,Y 237.421,Z 570.979,A -85,B 0,C 180,E1 -19717.655,E2 -19717.655} C_VEL
LIN {X 0,Y 239.273,Z 561.353,A -85,B 0,C 180,E1 -19720.15,E2 -19720.15} C_VEL
LIN {X 0,Y 241.173,Z 551.399,A -85,B 0,C 180,E1 -19722.197,E2 -19722.197} C_VEL
LIN {X 0,Y 243.019,Z 540.139,A -85,B 0,C 180,E1 -19724.016,E2 -19724.016} C_VEL
LIN {X 0,Y 244.489,Z 529.139,A -85,B 0,C 180,E1 -19725.42,E2 -19725.42} C_VEL
LIN {X 0,Y 245.879,Z 516.913,A -85,B 0,C 180,E1 -19726.608,E2 -19726.608} C_VEL
LIN {X 0,Y 246.944,Z 503.956,A -85,B 0,C 180,E1 -19727.494,E2 -19727.494} C_VEL
LIN {X 0,Y 247.541,Z 491.649,A -85,B 0,C 180,E1 -19728.037,E2 -19728.037} C_VEL
LIN {X 0,Y 249.589,Z 426.433,A -85,B 0,C 180,E1 -19729.872,E2 -19729.872} C_VEL
LIN {X 0,Y 243.744,Z 410.599,A -85,B 0,C 180,E1 -19731.041,E2 -19731.041} C_VEL
LIN {X 0,Y 237.424,Z 397.816,A -85,B 0,C 180,E1 -19732.236,E2 -19732.236} C_VEL
LIN {X 0,Y 235.201,Z 393.264,A -85,B 0,C 180,E1 -19732.677,E2 -19732.677} C_VEL
LIN {X 0,Y 234.974,Z 392.216,A -85,B 0,C 180,E1 -19732.747,E2 -19732.747} C_VEL
LIN {X 0,Y 234.974,Z 392.211,A -85,B 0,C 180,E1 -19736.656,E2 -19736.656} C_VEL
LIN {X 0,Y 234.935,Z 392.221,A -85,B 0,C 180,E1 -19740.566,E2 -19740.566} C_VEL
LIN {X 0,Y 234.943,Z 392.22,A -85,B 0,C 180,E1 -19744.635,E2 -19744.635} C_VEL
LIN {X 0,Y 234.942,Z 392.217,A -85,B 0,C 180,E1 -19748.943,E2 -19748.943} C_VEL
LIN {X 0,Y 234.923,Z 392.219,A -85,B 0,C 180,E1 -19753.477,E2 -19753.477} C_VEL
LIN {X 0,Y 234.974,Z 392.204,A -85,B 0,C 180,E1 -19756.533,E2 -19756.533} C_VEL
LIN {X 0,Y 234.954,Z 392.216,A -85,B 0,C 180,E1 -19761.085,E2 -19761.085} C_VEL
LIN {X 0,Y 234.959,Z 392.199,A -85,B 0,C 180,E1 -19765.366,E2 -19765.366} C_VEL
LIN {X 0,Y 234.921,Z 392.221,A -85,B 0,C 180,E1 -19769.43,E2 -19769.43} C_VEL
LIN {X 0,Y 234.991,Z 392.199,A -85,B 0,C 180,E1 -19773.793,E2 -19773.793} C_VEL
LIN {X 0,Y 235.024,Z 392.208,A -85,B 0,C 180,E1 -19778.97,E2 -19778.97} C_VEL
LIN {X 0,Y 235.093,Z 392.187,A -85,B 0,C 180,E1 -19783.058,E2 -19783.058} C_VEL
LIN {X 0,Y 235.114,Z 392.194,A -85,B 0,C 180,E1 -19787.921,E2 -19787.921} C_VEL
LIN {X 0,Y 235.372,Z 392.162,A -85,B 0,C 180,E1 -19791.413,E2 -19791.413} C_VEL
LIN {X 0,Y 235.399,Z 392.151,A -85,B 0,C 180,E1 -19793.141,E2 -19793.141} C_VEL
LIN {X 0,Y 235.591,Z 392.135,A -85,B 0,C 180,E1 -19798.29,E2 -19798.29} C_VEL
LIN {X 0,Y 235.592,Z 392.138,A -85,B 0,C 180,E1 -19801.709,E2 -19801.709} C_VEL
LIN {X 0,Y 235.399,Z 392.16,A -85,B 0,C 180,E1 -19806.858,E2 -19806.858} C_VEL
LIN {X 0,Y 235.233,Z 392.184,A -85,B 0,C 180,E1 -19810.326,E2 -19810.326} C_VEL
LIN {X 0,Y 235.107,Z 392.198,A -85,B 0,C 180,E1 -19815.606,E2 -19815.606} C_VEL
LIN {X 0,Y 235.015,Z 392.205,A -85,B 0,C 180,E1 -19819.205,E2 -19819.205} C_VEL
LIN {X 0,Y 234.976,Z 392.212,A -85,B 0,C 180,E1 -19822.881,E2 -19822.881} C_VEL
LIN {X 0,Y 234.971,Z 392.213,A -85,B 0,C 180,E1 -19824.552,E2 -19824.552} C_VEL
LIN {X 0,Y 234.359,Z 392.298,A -85,B 0,C 180,E1 -19825.984,E2 -19825.984} C_VEL
LIN {X 0,Y 232.787,Z 392.498,A -85,B 0,C 180,E1 -19827.389,E2 -19827.389} C_VEL
LIN {X 0,Y 229.012,Z 392.964,A -85,B 0,C 180,E1 -19830.22,E2 -19830.22} C_VEL
LIN {X 0,Y 227.935,Z 393.094,A -85,B 0,C 180,E1 -19831.698,E2 -19831.698} C_VEL
LIN {X 0,Y 227.843,Z 393.102,A -85,B 0,C 180,E1 -19832.2,E2 -19832.2} C_VEL
LIN {X 0,Y 227.905,Z 393.096,A -85,B 0,C 180,E1 -19836.702,E2 -19836.702} C_VEL
LIN {X 0,Y 227.889,Z 393.099,A -85,B 0,C 180,E1 -19840.363,E2 -19840.363} C_VEL
LIN {X 0,Y 227.906,Z 393.095,A -85,B 0,C 180,E1 -19842.72,E2 -19842.72} C_VEL
LIN {X 0,Y 227.887,Z 393.1,A -85,B 0,C 180,E1 -19847.744,E2 -19847.744} C_VEL
LIN {X 0,Y 227.935,Z 393.204,A -85,B 0,C 180,E1 -19851.528,E2 -19851.528} C_VEL
LIN {X 0,Y 230.09,Z 402.501,A -85,B 0,C 180,E1 -19855.558,E2 -19855.558} C_VEL
LIN {X 0,Y 231.212,Z 407.676,A -85,B 0,C 180,E1 -19857.65,E2 -19857.65} C_VEL
LIN {X 0,Y 237.979,Z 425.69,A -85,B 0,C 180,E1 -19859.123,E2 -19859.123} C_VEL
LIN {X 0,Y 242.108,Z 461.292,A -85,B 0,C 180,E1 -19860.769,E2 -19860.769} C_VEL
LIN {X 0,Y 241.976,Z 473.421,A -85,B 0,C 180,E1 -19861.145,E2 -19861.145} C_VEL
LIN {X 0,Y 240.398,Z 516.557,A -85,B 0,C 180,E1 -19862.408,E2 -19862.408} C_VEL
LIN {X 0,Y 239.413,Z 529.833,A -85,B 0,C 180,E1 -19863.112,E2 -19863.112} C_VEL
LIN {X 0,Y 238.018,Z 542.001,A -85,B 0,C 180,E1 -19864.064,E2 -19864.064} C_VEL
LIN {X 0,Y 236.253,Z 554.275,A -85,B 0,C 180,E1 -19865.389,E2 -19865.389} C_VEL
LIN {X 0,Y 234.226,Z 565.9,A -85,B 0,C 180,E1 -19867.042,E2 -19867.042} C_VEL
LIN {X 0,Y 232.21,Z 576.368,A -85,B 0,C 180,E1 -19868.937,E2 -19868.937} C_VEL
LIN {X 0,Y 230.539,Z 585.102,A -85,B 0,C 180,E1 -19870.915,E2 -19870.915} C_VEL
LIN {X 0,Y 229.161,Z 592.83,A -85,B 0,C 180,E1 -19873.062,E2 -19873.062} C_VEL
LIN {X 0,Y 227.718,Z 600.521,A -85,B 0,C 180,E1 -19875.706,E2 -19875.706} C_VEL
LIN {X 0,Y 226.639,Z 606.697,A -85,B 0,C 180,E1 -19878.372,E2 -19878.372} C_VEL
LIN {X 0,Y 226.07,Z 611.594,A -85,B 0,C 180,E1 -19881.058,E2 -19881.058} C_VEL
LIN {X 0,Y 225.764,Z 615.341,A -85,B 0,C 180,E1 -19883.745,E2 -19883.745} C_VEL
LIN {X 0,Y 225.752,Z 618.051,A -85,B 0,C 180,E1 -19886.43,E2 -19886.43} C_VEL
LIN {X 0,Y 225.862,Z 619.323,A -85,B 0,C 180,E1 -19888.217,E2 -19888.217} C_VEL
LIN {X 0,Y 225.878,Z 620.182,A -85,B 0,C 180,E1 -19890,E2 -19890} C_VEL
LIN {X 0,Y 225.831,Z 620.594,A -85,B 0,C 180,E1 -19891.783,E2 -19891.783} C_VEL
LIN {X 0,Y 225.684,Z 620.226,A -85,B 0,C 180,E1 -19895.36,E2 -19895.36} C_VEL
LIN {X 0,Y 225.768,Z 619.467,A -85,B 0,C 180,E1 -19897.153,E2 -19897.153} C_VEL
LIN {X 0,Y 226.054,Z 618.287,A -85,B 0,C 180,E1 -19898.943,E2 -19898.943} C_VEL
LIN {X 0,Y 226.825,Z 615.76,A -85,B 0,C 180,E1 -19901.618,E2 -19901.618} C_VEL
LIN {X 0,Y 227.939,Z 612.239,A -85,B 0,C 180,E1 -19904.28,E2 -19904.28} C_VEL
LIN {X 0,Y 229.755,Z 607.653,A -85,B 0,C 180,E1 -19906.893,E2 -19906.893} C_VEL
LIN {X 0,Y 232.315,Z 600.632,A -85,B 0,C 180,E1 -19909.94,E2 -19909.94} C_VEL
LIN {X 0,Y 234.836,Z 593.283,A -85,B 0,C 180,E1 -19912.431,E2 -19912.431} C_VEL
LIN {X 0,Y 237.445,Z 585.707,A -85,B 0,C 180,E1 -19914.48,E2 -19914.48} C_VEL
LIN {X 0,Y 240.481,Z 576.556,A -85,B 0,C 180,E1 -19916.466,E2 -19916.466} C_VEL
LIN {X 0,Y 243.457,Z 566.413,A -85,B 0,C 180,E1 -19918.209,E2 -19918.209} C_VEL
LIN {X 0,Y 246.303,Z 555.186,A -85,B 0,C 180,E1 -19919.72,E2 -19919.72} C_VEL
LIN {X 0,Y 249.033,Z 542.567,A -85,B 0,C 180,E1 -19920.999,E2 -19920.999} C_VEL
LIN {X 0,Y 251.094,Z 530.247,A -85,B 0,C 180,E1 -19921.89,E2 -19921.89} C_VEL
LIN {X 0,Y 252.537,Z 516.812,A -85,B 0,C 180,E1 -19922.559,E2 -19922.559} C_VEL
LIN {X 0,Y 254.2,Z 483.318,A -85,B 0,C 180,E1 -19923.509,E2 -19923.509} C_VEL
LIN {X 0,Y 254.893,Z 466.956,A -85,B 0,C 180,E1 -19923.961,E2 -19923.961} C_VEL
LIN {X 0,Y 251.796,Z 446.065,A -85,B 0,C 180,E1 -19925.248,E2 -19925.248} C_VEL
LIN {X 0,Y 244.872,Z 430.728,A -85,B 0,C 180,E1 -19927.14,E2 -19927.14} C_VEL
LIN {X 0,Y 238.837,Z 419.086,A -85,B 0,C 180,E1 -19928.859,E2 -19928.859} C_VEL
LIN {X 0,Y 236.174,Z 414.337,A -85,B 0,C 180,E1 -19929.646,E2 -19929.646} C_VEL
LIN {X 0,Y 233.626,Z 409.898,A -85,B 0,C 180,E1 -19930.422,E2 -19930.422} C_VEL
LIN {X 0,Y 231.477,Z 405.865,A -85,B 0,C 180,E1 -19931.138,E2 -19931.138} C_VEL
LIN {X 0,Y 229.405,Z 398.498,A -85,B 0,C 180,E1 -19935.201,E2 -19935.201} C_VEL
LIN {X 0,Y 227.913,Z 393.088,A -85,B 0,C 180,E1 -19938.448,E2 -19938.448} C_VEL
LIN {X 0,Y 227.905,Z 393.092,A -85,B 0,C 180,E1 -19943.298,E2 -19943.298} C_VEL
LIN {X 0,Y 227.887,Z 393.098,A -85,B 0,C 180,E1 -19946.373,E2 -19946.373} C_VEL
LIN {X 0,Y 227.915,Z 393.09,A -85,B 0,C 180,E1 -19950.438,E2 -19950.438} C_VEL
LIN {X 0,Y 227.924,Z 393.06,A -85,B 0,C 180,E1 -19954.426,E2 -19954.426} C_VEL
LIN {X 0,Y 227.958,Z 393.089,A -85,B 0,C 180,E1 -19958.287,E2 -19958.287} C_VEL
LIN {X 0,Y 228.03,Z 393.081,A -85,B 0,C 180,E1 -19962.826,E2 -19962.826} C_VEL
LIN {X 0,Y 228.088,Z 393.073,A -85,B 0,C 180,E1 -19967.544,E2 -19967.544} C_VEL
LIN {X 0,Y 228.301,Z 393.045,A -85,B 0,C 180,E1 -19971.146,E2 -19971.146} C_VEL
LIN {X 0,Y 228.35,Z 393.034,A -85,B 0,C 180,E1 -19972.929,E2 -19972.929} C_VEL
LIN {X 0,Y 228.55,Z 393.006,A -85,B 0,C 180,E1 -19978.238,E2 -19978.238} C_VEL
LIN {X 0,Y 228.55,Z 393.015,A -85,B 0,C 180,E1 -19981.763,E2 -19981.763} C_VEL
LIN {X 0,Y 228.319,Z 393.038,A -85,B 0,C 180,E1 -19987.073,E2 -19987.073} C_VEL
LIN {X 0,Y 228.141,Z 393.068,A -85,B 0,C 180,E1 -19990.652,E2 -19990.652} C_VEL
LIN {X 0,Y 228.056,Z 393.076,A -85,B 0,C 180,E1 -19994.273,E2 -19994.273} C_VEL
LIN {X 0,Y 227.999,Z 393.079,A -85,B 0,C 180,E1 -19997.954,E2 -19997.954} C_VEL
LIN {X 0,Y 227.927,Z 393.092,A -85,B 0,C 180,E1 -20002.33,E2 -20002.33} C_VEL
LIN {X 0,Y 227.94,Z 393.059,A -85,B 0,C 180,E1 -20006.604,E2 -20006.604} C_VEL
LIN {X 0,Y 227.906,Z 393.094,A -85,B 0,C 180,E1 -20010.297,E2 -20010.297} C_VEL
LIN {X 0,Y 227.888,Z 393.095,A -85,B 0,C 180,E1 -20013.719,E2 -20013.719} C_VEL
LIN {X 0,Y 227.87,Z 393.105,A -85,B 0,C 180,E1 -20018.087,E2 -20018.087} C_VEL
LIN {X 0,Y 227.937,Z 393.101,A -85,B 0,C 180,E1 -20019.122,E2 -20019.122} C_VEL
LIN {X 0,Y 228.817,Z 395.763,A -85,B 0,C 180,E1 -20019.469,E2 -20019.469} C_VEL
LIN {X 0,Y 231.147,Z 398.481,A -85,B 0,C 180,E1 -20020.178,E2 -20020.178} C_VEL
LIN {X 0,Y 233.33,Z 401.888,A -85,B 0,C 180,E1 -20020.858,E2 -20020.858} C_VEL
LIN {X 0,Y 234.734,Z 403.905,A -85,B 0,C 180,E1 -20021.277,E2 -20021.277} C_VEL
LIN {X 0,Y 241.955,Z 414.855,A -85,B 0,C 180,E1 -20023.333,E2 -20023.333} C_VEL
LIN {X 0,Y 247.261,Z 423.833,A -85,B 0,C 180,E1 -20024.764,E2 -20024.764} C_VEL
LIN {X 0,Y 254.394,Z 438.546,A -85,B 0,C 180,E1 -20026.641,E2 -20026.641} C_VEL
LIN {X 0,Y 255.945,Z 442,A -85,B 0,C 180,E1 -20027.038,E2 -20027.038} C_VEL
LIN {X 0,Y 253.392,Z 496.843,A -85,B 0,C 180,E1 -20028.568,E2 -20028.568} C_VEL
LIN {X 0,Y 252.174,Z 509.414,A -85,B 0,C 180,E1 -20029.189,E2 -20029.189} C_VEL
LIN {X 0,Y 250.394,Z 522.679,A -85,B 0,C 180,E1 -20030.187,E2 -20030.187} C_VEL
LIN {X 0,Y 247.891,Z 534.808,A -85,B 0,C 180,E1 -20031.412,E2 -20031.412} C_VEL
LIN {X 0,Y 245.63,Z 545.092,A -85,B 0,C 180,E1 -20032.813,E2 -20032.813} C_VEL
LIN {X 0,Y 242.877,Z 555.724,A -85,B 0,C 180,E1 -20034.64,E2 -20034.64} C_VEL
LIN {X 0,Y 239.881,Z 565.212,A -85,B 0,C 180,E1 -20036.68,E2 -20036.68} C_VEL
LIN {X 0,Y 236.696,Z 574.462,A -85,B 0,C 180,E1 -20039.241,E2 -20039.241} C_VEL
LIN {X 0,Y 234.035,Z 581.622,A -85,B 0,C 180,E1 -20041.774,E2 -20041.774} C_VEL
LIN {X 0,Y 232.044,Z 586.51,A -85,B 0,C 180,E1 -20043.95,E2 -20043.95} C_VEL
LIN {X 0,Y 230.022,Z 591.226,A -85,B 0,C 180,E1 -20046.598,E2 -20046.598} C_VEL
LIN {X 0,Y 228.477,Z 594.794,A -85,B 0,C 180,E1 -20049.284,E2 -20049.284} C_VEL
LIN {X 0,Y 227.319,Z 597.318,A -85,B 0,C 180,E1 -20051.991,E2 -20051.991} C_VEL
LIN {X 0,Y 226.702,Z 598.55,A -85,B 0,C 180,E1 -20053.955,E2 -20053.955} C_VEL
LIN {X 0,Y 225.933,Z 599.51,A -85,B 0,C 180,E1 -20057.424,E2 -20057.424} C_VEL
LIN {X 0,Y 225.733,Z 599.442,A -85,B 0,C 180,E1 -20059.234,E2 -20059.234} C_VEL
LIN {X 0,Y 225.675,Z 598.974,A -85,B 0,C 180,E1 -20061.042,E2 -20061.042} C_VEL
LIN {X 0,Y 225.96,Z 596.935,A -85,B 0,C 180,E1 -20064.445,E2 -20064.445} C_VEL
LIN {X 0,Y 226.215,Z 594.058,A -85,B 0,C 180,E1 -20067.329,E2 -20067.329} C_VEL
LIN {X 0,Y 226.832,Z 590.33,A -85,B 0,C 180,E1 -20070,E2 -20070} C_VEL
LIN {X 0,Y 227.62,Z 585.503,A -85,B 0,C 180,E1 -20072.654,E2 -20072.654} C_VEL
LIN {X 0,Y 228.817,Z 579.417,A -85,B 0,C 180,E1 -20075.287,E2 -20075.287} C_VEL
LIN {X 0,Y 230.401,Z 571.852,A -85,B 0,C 180,E1 -20077.889,E2 -20077.889} C_VEL
LIN {X 0,Y 232.004,Z 564.111,A -85,B 0,C 180,E1 -20080.031,E2 -20080.031} C_VEL
LIN {X 0,Y 234.065,Z 553.597,A -85,B 0,C 180,E1 -20082.353,E2 -20082.353} C_VEL
LIN {X 0,Y 235.938,Z 542.903,A -85,B 0,C 180,E1 -20084.226,E2 -20084.226} C_VEL
LIN {X 0,Y 237.519,Z 532.514,A -85,B 0,C 180,E1 -20085.664,E2 -20085.664} C_VEL
LIN {X 0,Y 239.005,Z 520.055,A -85,B 0,C 180,E1 -20086.99,E2 -20086.99} C_VEL
LIN {X 0,Y 240.258,Z 506.88,A -85,B 0,C 180,E1 -20087.997,E2 -20087.997} C_VEL
LIN {X 0,Y 240.901,Z 494.95,A -85,B 0,C 180,E1 -20088.607,E2 -20088.607} C_VEL
LIN {X 0,Y 243.175,Z 427.975,A -85,B 0,C 180,E1 -20090.545,E2 -20090.545} C_VEL
LIN {X 0,Y 237.27,Z 412.348,A -85,B 0,C 180,E1 -20091.768,E2 -20091.768} C_VEL
LIN {X 0,Y 230.691,Z 399.198,A -85,B 0,C 180,E1 -20093.073,E2 -20093.073} C_VEL
LIN {X 0,Y 228.093,Z 394.063,A -85,B 0,C 180,E1 -20093.612,E2 -20093.612} C_VEL
LIN {X 0,Y 227.901,Z 393.097,A -85,B 0,C 180,E1 -20093.694,E2 -20093.694} C_VEL
LIN {X 0,Y 227.891,Z 393.097,A -85,B 0,C 180,E1 -20097.554,E2 -20097.554} C_VEL
LIN {X 0,Y 227.874,Z 393.099,A -85,B 0,C 180,E1 -20101.621,E2 -20101.621} C_VEL
LIN {X 0,Y 227.884,Z 393.099,A -85,B 0,C 180,E1 -20105.87,E2 -20105.87} C_VEL
LIN {X 0,Y 227.828,Z 393.097,A -85,B 0,C 180,E1 -20110.375,E2 -20110.375} C_VEL
LIN {X 0,Y 227.86,Z 393.097,A -85,B 0,C 180,E1 -20115.185,E2 -20115.185} C_VEL
LIN {X 0,Y 227.917,Z 393.08,A -85,B 0,C 180,E1 -20117.735,E2 -20117.735} C_VEL
LIN {X 0,Y 227.87,Z 393.1,A -85,B 0,C 180,E1 -20121.913,E2 -20121.913} C_VEL
LIN {X 0,Y 227.888,Z 393.085,A -85,B 0,C 180,E1 -20126.372,E2 -20126.372} C_VEL
LIN {X 0,Y 227.902,Z 393.096,A -85,B 0,C 180,E1 -20130.435,E2 -20130.435} C_VEL
LIN {X 0,Y 227.926,Z 393.076,A -85,B 0,C 180,E1 -20134.425,E2 -20134.425} C_VEL
LIN {X 0,Y 227.988,Z 393.086,A -85,B 0,C 180,E1 -20138.289,E2 -20138.289} C_VEL
LIN {X 0,Y 228.032,Z 393.067,A -85,B 0,C 180,E1 -20142.824,E2 -20142.824} C_VEL
LIN {X 0,Y 228.07,Z 393.069,A -85,B 0,C 180,E1 -20147.543,E2 -20147.543} C_VEL
LIN {X 0,Y 228.302,Z 393.043,A -85,B 0,C 180,E1 -20151.145,E2 -20151.145} C_VEL
LIN {X 0,Y 228.35,Z 393.029,A -85,B 0,C 180,E1 -20152.928,E2 -20152.928} C_VEL
LIN {X 0,Y 228.55,Z 393.011,A -85,B 0,C 180,E1 -20158.237,E2 -20158.237} C_VEL
LIN {X 0,Y 228.55,Z 393.015,A -85,B 0,C 180,E1 -20161.762,E2 -20161.762} C_VEL
LIN {X 0,Y 228.35,Z 393.038,A -85,B 0,C 180,E1 -20167.071,E2 -20167.071} C_VEL
LIN {X 0,Y 228.159,Z 393.064,A -85,B 0,C 180,E1 -20170.65,E2 -20170.65} C_VEL
LIN {X 0,Y 228.058,Z 393.074,A -85,B 0,C 180,E1 -20174.272,E2 -20174.272} C_VEL
LIN {X 0,Y 228.002,Z 393.082,A -85,B 0,C 180,E1 -20177.953,E2 -20177.953} C_VEL
LIN {X 0,Y 227.956,Z 393.089,A -85,B 0,C 180,E1 -20182.348,E2 -20182.348} C_VEL
LIN {X 0,Y 227.938,Z 393.092,A -85,B 0,C 180,E1 -20186.602,E2 -20186.602} C_VEL
LIN {X 0,Y 227.893,Z 393.099,A -85,B 0,C 180,E1 -20190.291,E2 -20190.291} C_VEL
LIN {X 0,Y 227.843,Z 393.102,A -85,B 0,C 180,E1 -20192.2,E2 -20192.2} C_VEL
LIN {X 0,Y 227.166,Z 393.19,A -85,B 0,C 180,E1 -20193.677,E2 -20193.677} C_VEL
LIN {X 0,Y 224.33,Z 393.544,A -85,B 0,C 180,E1 -20196.087,E2 -20196.087} C_VEL
LIN {X 0,Y 221.936,Z 393.841,A -85,B 0,C 180,E1 -20198.054,E2 -20198.054} C_VEL
LIN {X 0,Y 220.923,Z 393.967,A -85,B 0,C 180,E1 -20199.58,E2 -20199.58} C_VEL
LIN {X 0,Y 220.848,Z 393.976,A -85,B 0,C 180,E1 -20200.097,E2 -20200.097} C_VEL
LIN {X 0,Y 220.827,Z 393.976,A -85,B 0,C 180,E1 -20204.44,E2 -20204.44} C_VEL
LIN {X 0,Y 220.829,Z 393.981,A -85,B 0,C 180,E1 -20208.062,E2 -20208.062} C_VEL
LIN {X 0,Y 220.852,Z 394.026,A -85,B 0,C 180,E1 -20210.76,E2 -20210.76} C_VEL
LIN {X 0,Y 222.662,Z 401.563,A -85,B 0,C 180,E1 -20214.201,E2 -20214.201} C_VEL
LIN {X 0,Y 223.97,Z 407.428,A -85,B 0,C 180,E1 -20216.642,E2 -20216.642} C_VEL
LIN {X 0,Y 231.7,Z 427.214,A -85,B 0,C 180,E1 -20218.389,E2 -20218.389} C_VEL
LIN {X 0,Y 235.704,Z 462.046,A -85,B 0,C 180,E1 -20220.06,E2 -20220.06} C_VEL
LIN {X 0,Y 235.539,Z 473.515,A -85,B 0,C 180,E1 -20220.422,E2 -20220.422} C_VEL
LIN {X 0,Y 233.939,Z 516.118,A -85,B 0,C 180,E1 -20221.7,E2 -20221.7} C_VEL
LIN {X 0,Y 232.926,Z 529.435,A -85,B 0,C 180,E1 -20222.422,E2 -20222.422} C_VEL
LIN {X 0,Y 231.475,Z 541.621,A -85,B 0,C 180,E1 -20223.396,E2 -20223.396} C_VEL
LIN {X 0,Y 229.802,Z 553.108,A -85,B 0,C 180,E1 -20224.65,E2 -20224.65} C_VEL
LIN {X 0,Y 227.605,Z 564.881,A -85,B 0,C 180,E1 -20226.334,E2 -20226.334} C_VEL
LIN {X 0,Y 225.5,Z 575.469,A -85,B 0,C 180,E1 -20228.279,E2 -20228.279} C_VEL
LIN {X 0,Y 223.609,Z 585.193,A -85,B 0,C 180,E1 -20230.543,E2 -20230.543} C_VEL
LIN {X 0,Y 222.36,Z 592.127,A -85,B 0,C 180,E1 -20232.527,E2 -20232.527} C_VEL
LIN {X 0,Y 220.796,Z 599.896,A -85,B 0,C 180,E1 -20235.248,E2 -20235.248} C_VEL
LIN {X 0,Y 219.644,Z 606.127,A -85,B 0,C 180,E1 -20237.996,E2 -20237.996} C_VEL
LIN {X 0,Y 219.023,Z 611.075,A -85,B 0,C 180,E1 -20240.768,E2 -20240.768} C_VEL
LIN {X 0,Y 218.699,Z 614.87,A -85,B 0,C 180,E1 -20243.542,E2 -20243.542} C_VEL
LIN {X 0,Y 218.66,Z 617.623,A -85,B 0,C 180,E1 -20246.314,E2 -20246.314} C_VEL
LIN {X 0,Y 218.767,Z 618.917,A -85,B 0,C 180,E1 -20248.159,E2 -20248.159} C_VEL
LIN {X 0,Y 218.809,Z 619.801,A -85,B 0,C 180,E1 -20250,E2 -20250} C_VEL
LIN {X 0,Y 218.737,Z 620.25,A -85,B 0,C 180,E1 -20251.841,E2 -20251.841} C_VEL
LIN {X 0,Y 218.587,Z 619.921,A -85,B 0,C 180,E1 -20255.535,E2 -20255.535} C_VEL
LIN {X 0,Y 219.018,Z 618.044,A -85,B 0,C 180,E1 -20259.232,E2 -20259.232} C_VEL
LIN {X 0,Y 219.53,Z 616.467,A -85,B 0,C 180,E1 -20261.074,E2 -20261.074} C_VEL
LIN {X 0,Y 220.568,Z 613.329,A -85,B 0,C 180,E1 -20263.826,E2 -20263.826} C_VEL
LIN {X 0,Y 222.269,Z 609.16,A -85,B 0,C 180,E1 -20266.533,E2 -20266.533} C_VEL
LIN {X 0,Y 224.791,Z 602.827,A -85,B 0,C 180,E1 -20269.639,E2 -20269.639} C_VEL
LIN {X 0,Y 227.325,Z 595.962,A -85,B 0,C 180,E1 -20272.254,E2 -20272.254} C_VEL
LIN {X 0,Y 229.86,Z 588.981,A -85,B 0,C 180,E1 -20274.378,E2 -20274.378} C_VEL
LIN {X 0,Y 232.925,Z 580.599,A -85,B 0,C 180,E1 -20276.426,E2 -20276.426} C_VEL
LIN {X 0,Y 235.894,Z 571.455,A -85,B 0,C 180,E1 -20278.226,E2 -20278.226} C_VEL
LIN {X 0,Y 238.711,Z 561.538,A -85,B 0,C 180,E1 -20279.789,E2 -20279.789} C_VEL
LIN {X 0,Y 241.387,Z 550.78,A -85,B 0,C 180,E1 -20281.117,E2 -20281.117} C_VEL
LIN {X 0,Y 243.833,Z 538.948,A -85,B 0,C 180,E1 -20282.223,E2 -20282.223} C_VEL
LIN {X 0,Y 245.824,Z 526.183,A -85,B 0,C 180,E1 -20283.087,E2 -20283.087} C_VEL
LIN {X 0,Y 247.158,Z 512.707,A -85,B 0,C 180,E1 -20283.664,E2 -20283.664} C_VEL
LIN {X 0,Y 249.186,Z 467.563,A -85,B 0,C 180,E1 -20284.949,E2 -20284.949} C_VEL
LIN {X 0,Y 246.457,Z 448.906,A -85,B 0,C 180,E1 -20286.144,E2 -20286.144} C_VEL
LIN {X 0,Y 239.486,Z 433.311,A -85,B 0,C 180,E1 -20288.154,E2 -20288.154} C_VEL
LIN {X 0,Y 232.858,Z 420.514,A -85,B 0,C 180,E1 -20290.157,E2 -20290.157} C_VEL
LIN {X 0,Y 226.772,Z 410.109,A -85,B 0,C 180,E1 -20292.11,E2 -20292.11} C_VEL
LIN {X 0,Y 224.241,Z 405.713,A -85,B 0,C 180,E1 -20292.979,E2 -20292.979} C_VEL
LIN {X 0,Y 222.127,Z 398.411,A -85,B 0,C 180,E1 -20297.19,E2 -20297.19} C_VEL
LIN {X 0,Y 220.846,Z 393.969,A -85,B 0,C 180,E1 -20300.076,E2 -20300.076} C_VEL
LIN {X 0,Y 220.831,Z 393.972,A -85,B 0,C 180,E1 -20302.795,E2 -20302.795} C_VEL
LIN {X 0,Y 220.821,Z 393.977,A -85,B 0,C 180,E1 -20307.245,E2 -20307.245} C_VEL
LIN {X 0,Y 220.833,Z 393.979,A -85,B 0,C 180,E1 -20311.486,E2 -20311.486} C_VEL
LIN {X 0,Y 220.863,Z 393.938,A -85,B 0,C 180,E1 -20315.565,E2 -20315.565} C_VEL
LIN {X 0,Y 220.888,Z 393.967,A -85,B 0,C 180,E1 -20319.514,E2 -20319.514} C_VEL
LIN {X 0,Y 221.011,Z 393.953,A -85,B 0,C 180,E1 -20323.37,E2 -20323.37} C_VEL
LIN {X 0,Y 221.107,Z 393.933,A -85,B 0,C 180,E1 -20329.006,E2 -20329.006} C_VEL
LIN {X 0,Y 221.301,Z 393.914,A -85,B 0,C 180,E1 -20332.702,E2 -20332.702} C_VEL
LIN {X 0,Y 221.508,Z 393.883,A -85,B 0,C 180,E1 -20338.182,E2 -20338.182} C_VEL
LIN {X 0,Y 221.508,Z 393.892,A -85,B 0,C 180,E1 -20341.819,E2 -20341.819} C_VEL
LIN {X 0,Y 221.255,Z 393.916,A -85,B 0,C 180,E1 -20347.3,E2 -20347.3} C_VEL
LIN {X 0,Y 221.063,Z 393.947,A -85,B 0,C 180,E1 -20350.997,E2 -20350.997} C_VEL
LIN {X 0,Y 221.011,Z 393.946,A -85,B 0,C 180,E1 -20356.631,E2 -20356.631} C_VEL
LIN {X 0,Y 220.889,Z 393.962,A -85,B 0,C 180,E1 -20360.487,E2 -20360.487} C_VEL
LIN {X 0,Y 220.864,Z 393.956,A -85,B 0,C 180,E1 -20364.436,E2 -20364.436} C_VEL
LIN {X 0,Y 220.834,Z 393.962,A -85,B 0,C 180,E1 -20368.515,E2 -20368.515} C_VEL
LIN {X 0,Y 220.822,Z 393.98,A -85,B 0,C 180,E1 -20372.756,E2 -20372.756} C_VEL
LIN {X 0,Y 220.833,Z 393.975,A -85,B 0,C 180,E1 -20377.206,E2 -20377.206} C_VEL
LIN {X 0,Y 221.622,Z 396.422,A -85,B 0,C 180,E1 -20377.55,E2 -20377.55} C_VEL
LIN {X 0,Y 223.473,Z 398.675,A -85,B 0,C 180,E1 -20378.175,E2 -20378.175} C_VEL
LIN {X 0,Y 224.362,Z 399.708,A -85,B 0,C 180,E1 -20378.467,E2 -20378.467} C_VEL
LIN {X 0,Y 226.541,Z 402.95,A -85,B 0,C 180,E1 -20379.197,E2 -20379.197} C_VEL
LIN {X 0,Y 228.158,Z 405.314,A -85,B 0,C 180,E1 -20379.722,E2 -20379.722} C_VEL
LIN {X 0,Y 232.721,Z 411.809,A -85,B 0,C 180,E1 -20381.132,E2 -20381.132} C_VEL
LIN {X 0,Y 241.357,Z 425.664,A -85,B 0,C 180,E1 -20383.63,E2 -20383.63} C_VEL
LIN {X 0,Y 248.376,Z 439.908,A -85,B 0,C 180,E1 -20385.579,E2 -20385.579} C_VEL
LIN {X 0,Y 250.264,Z 444.136,A -85,B 0,C 180,E1 -20386.089,E2 -20386.089} C_VEL
LIN {X 0,Y 247.711,Z 496.978,A -85,B 0,C 180,E1 -20387.588,E2 -20387.588} C_VEL
LIN {X 0,Y 246.421,Z 509.959,A -85,B 0,C 180,E1 -20388.243,E2 -20388.243} C_VEL
LIN {X 0,Y 244.687,Z 522.479,A -85,B 0,C 180,E1 -20389.2,E2 -20389.2} C_VEL
LIN {X 0,Y 242.311,Z 533.967,A -85,B 0,C 180,E1 -20390.352,E2 -20390.352} C_VEL
LIN {X 0,Y 239.857,Z 544.459,A -85,B 0,C 180,E1 -20391.759,E2 -20391.759} C_VEL
LIN {X 0,Y 237.016,Z 555.262,A -85,B 0,C 180,E1 -20393.628,E2 -20393.628} C_VEL
LIN {X 0,Y 233.845,Z 564.925,A -85,B 0,C 180,E1 -20395.702,E2 -20395.702} C_VEL
LIN {X 0,Y 230.53,Z 574.156,A -85,B 0,C 180,E1 -20398.273,E2 -20398.273} C_VEL
LIN {X 0,Y 227.664,Z 581.544,A -85,B 0,C 180,E1 -20400.909,E2 -20400.909} C_VEL
LIN {X 0,Y 225.535,Z 586.511,A -85,B 0,C 180,E1 -20403.139,E2 -20403.139} C_VEL
LIN {X 0,Y 223.392,Z 591.299,A -85,B 0,C 180,E1 -20405.859,E2 -20405.859} C_VEL
LIN {X 0,Y 221.686,Z 594.935,A -85,B 0,C 180,E1 -20408.619,E2 -20408.619} C_VEL
LIN {X 0,Y 220.434,Z 597.521,A -85,B 0,C 180,E1 -20411.409,E2 -20411.409} C_VEL
LIN {X 0,Y 219.68,Z 598.922,A -85,B 0,C 180,E1 -20413.693,E2 -20413.693} C_VEL
LIN {X 0,Y 218.896,Z 599.833,A -85,B 0,C 180,E1 -20417.012,E2 -20417.012} C_VEL
LIN {X 0,Y 218.6,Z 599.368,A -85,B 0,C 180,E1 -20420.75,E2 -20420.75} C_VEL
LIN {X 0,Y 218.647,Z 598.51,A -85,B 0,C 180,E1 -20422.613,E2 -20422.613} C_VEL
LIN {X 0,Y 218.889,Z 597.239,A -85,B 0,C 180,E1 -20424.473,E2 -20424.473} C_VEL
LIN {X 0,Y 219.126,Z 594.588,A -85,B 0,C 180,E1 -20427.243,E2 -20427.243} C_VEL
LIN {X 0,Y 219.718,Z 590.929,A -85,B 0,C 180,E1 -20430,E2 -20430} C_VEL
LIN {X 0,Y 220.557,Z 586.169,A -85,B 0,C 180,E1 -20432.74,E2 -20432.74} C_VEL
LIN {X 0,Y 221.763,Z 580.162,A -85,B 0,C 180,E1 -20435.455,E2 -20435.455} C_VEL
LIN {X 0,Y 223.39,Z 572.688,A -85,B 0,C 180,E1 -20438.139,E2 -20438.139} C_VEL
LIN {X 0,Y 225.047,Z 565.058,A -85,B 0,C 180,E1 -20440.344,E2 -20440.344} C_VEL
LIN {X 0,Y 226.956,Z 555.778,A -85,B 0,C 180,E1 -20442.519,E2 -20442.519} C_VEL
LIN {X 0,Y 228.871,Z 545.465,A -85,B 0,C 180,E1 -20444.447,E2 -20444.447} C_VEL
LIN {X 0,Y 230.747,Z 534.021,A -85,B 0,C 180,E1 -20446.136,E2 -20446.136} C_VEL
LIN {X 0,Y 232.275,Z 522.033,A -85,B 0,C 180,E1 -20447.498,E2 -20447.498} C_VEL
LIN {X 0,Y 233.645,Z 508.672,A -85,B 0,C 180,E1 -20448.581,E2 -20448.581} C_VEL
LIN {X 0,Y 234.43,Z 495.266,A -85,B 0,C 180,E1 -20449.309,E2 -20449.309} C_VEL
LIN {X 0,Y 236.818,Z 429.698,A -85,B 0,C 180,E1 -20451.243,E2 -20451.243} C_VEL
LIN {X 0,Y 231.607,Z 415.878,A -85,B 0,C 180,E1 -20452.373,E2 -20452.373} C_VEL
LIN {X 0,Y 224.822,Z 402.26,A -85,B 0,C 180,E1 -20453.782,E2 -20453.782} C_VEL
LIN {X 0,Y 221.131,Z 394.985,A -85,B 0,C 180,E1 -20454.587,E2 -20454.587} C_VEL
LIN {X 0,Y 220.923,Z 393.955,A -85,B 0,C 180,E1 -20454.678,E2 -20454.678} C_VEL
LIN {X 0,Y 220.841,Z 393.974,A -85,B 0,C 180,E1 -20458.512,E2 -20458.512} C_VEL
LIN {X 0,Y 220.822,Z 393.979,A -85,B 0,C 180,E1 -20462.754,E2 -20462.754} C_VEL
LIN {X 0,Y 220.812,Z 393.978,A -85,B 0,C 180,E1 -20467.277,E2 -20467.277} C_VEL
LIN {X 0,Y 220.782,Z 393.974,A -85,B 0,C 180,E1 -20471.949,E2 -20471.949} C_VEL
LIN {X 0,Y 220.872,Z 393.957,A -85,B 0,C 180,E1 -20477.04,E2 -20477.04} C_VEL
LIN {X 0,Y 220.857,Z 393.974,A -85,B 0,C 180,E1 -20480.473,E2 -20480.473} C_VEL
LIN {X 0,Y 220.814,Z 393.96,A -85,B 0,C 180,E1 -20485.047,E2 -20485.047} C_VEL
LIN {X 0,Y 220.832,Z 393.976,A -85,B 0,C 180,E1 -20489.389,E2 -20489.389} C_VEL
LIN {X 0,Y 220.892,Z 393.954,A -85,B 0,C 180,E1 -20493.548,E2 -20493.548} C_VEL
LIN {X 0,Y 220.921,Z 393.961,A -85,B 0,C 180,E1 -20497.557,E2 -20497.557} C_VEL
LIN {X 0,Y 220.982,Z 393.945,A -85,B 0,C 180,E1 -20502.57,E2 -20502.57} C_VEL
LIN {X 0,Y 221.009,Z 393.948,A -85,B 0,C 180,E1 -20507.138,E2 -20507.138} C_VEL
LIN {X 0,Y 221.232,Z 393.924,A -85,B 0,C 180,E1 -20510.86,E2 -20510.86} C_VEL
LIN {X 0,Y 221.285,Z 393.909,A -85,B 0,C 180,E1 -20512.701,E2 -20512.701} C_VEL
LIN {X 0,Y 221.508,Z 393.887,A -85,B 0,C 180,E1 -20518.181,E2 -20518.181} C_VEL
LIN {X 0,Y 221.508,Z 393.892,A -85,B 0,C 180,E1 -20521.818,E2 -20521.818} C_VEL
LIN {X 0,Y 221.285,Z 393.918,A -85,B 0,C 180,E1 -20527.298,E2 -20527.298} C_VEL
LIN {X 0,Y 221.107,Z 393.942,A -85,B 0,C 180,E1 -20530.994,E2 -20530.994} C_VEL
LIN {X 0,Y 221.012,Z 393.954,A -85,B 0,C 180,E1 -20536.63,E2 -20536.63} C_VEL
LIN {X 0,Y 220.905,Z 393.969,A -85,B 0,C 180,E1 -20540.485,E2 -20540.485} C_VEL
LIN {X 0,Y 220.868,Z 393.972,A -85,B 0,C 180,E1 -20544.435,E2 -20544.435} C_VEL
LIN {X 0,Y 220.823,Z 393.977,A -85,B 0,C 180,E1 -20548.515,E2 -20548.515} C_VEL
LIN {X 0,Y 220.819,Z 393.979,A -85,B 0,C 180,E1 -20552.755,E2 -20552.755} C_VEL
LIN {X 0,Y 220.835,Z 393.977,A -85,B 0,C 180,E1 -20557.288,E2 -20557.288} C_VEL
LIN {X 0,Y 220.848,Z 393.976,A -85,B 0,C 180,E1 -20560.097,E2 -20560.097} C_VEL
LIN {X 0,Y 220.179,Z 394.061,A -85,B 0,C 180,E1 -20561.617,E2 -20561.617} C_VEL
LIN {X 0,Y 217.274,Z 394.42,A -85,B 0,C 180,E1 -20564.095,E2 -20564.095} C_VEL
LIN {X 0,Y 214.813,Z 394.73,A -85,B 0,C 180,E1 -20566.12,E2 -20566.12} C_VEL
LIN {X 0,Y 213.783,Z 394.856,A -85,B 0,C 180,E1 -20567.694,E2 -20567.694} C_VEL
LIN {X 0,Y 213.714,Z 394.861,A -85,B 0,C 180,E1 -20568.228,E2 -20568.228} C_VEL
LIN {X 0,Y 213.77,Z 394.9,A -85,B 0,C 180,E1 -20569.962,E2 -20569.962} C_VEL
LIN {X 0,Y 216.042,Z 404.322,A -85,B 0,C 180,E1 -20574.416,E2 -20574.416} C_VEL
LIN {X 0,Y 216.575,Z 406.805,A -85,B 0,C 180,E1 -20575.519,E2 -20575.519} C_VEL
LIN {X 0,Y 223.819,Z 424.68,A -85,B 0,C 180,E1 -20577.242,E2 -20577.242} C_VEL
LIN {X 0,Y 225.695,Z 430.016,A -85,B 0,C 180,E1 -20577.691,E2 -20577.691} C_VEL
LIN {X 0,Y 229.46,Z 464.63,A -85,B 0,C 180,E1 -20579.392,E2 -20579.392} C_VEL
LIN {X 0,Y 227.522,Z 515.652,A -85,B 0,C 180,E1 -20580.953,E2 -20580.953} C_VEL
LIN {X 0,Y 226.461,Z 529.011,A -85,B 0,C 180,E1 -20581.691,E2 -20581.691} C_VEL
LIN {X 0,Y 224.958,Z 541.22,A -85,B 0,C 180,E1 -20582.687,E2 -20582.687} C_VEL
LIN {X 0,Y 223.074,Z 553.533,A -85,B 0,C 180,E1 -20584.079,E2 -20584.079} C_VEL
LIN {X 0,Y 220.818,Z 565.162,A -85,B 0,C 180,E1 -20585.81,E2 -20585.81} C_VEL
LIN {X 0,Y 218.653,Z 575.645,A -85,B 0,C 180,E1 -20587.811,E2 -20587.811} C_VEL
LIN {X 0,Y 216.697,Z 585.243,A -85,B 0,C 180,E1 -20590.142,E2 -20590.142} C_VEL
LIN {X 0,Y 215.211,Z 592.824,A -85,B 0,C 180,E1 -20592.418,E2 -20592.418} C_VEL
LIN {X 0,Y 213.651,Z 600.396,A -85,B 0,C 180,E1 -20595.231,E2 -20595.231} C_VEL
LIN {X 0,Y 212.377,Z 607.38,A -85,B 0,C 180,E1 -20598.548,E2 -20598.548} C_VEL
LIN {X 0,Y 211.829,Z 611.98,A -85,B 0,C 180,E1 -20601.414,E2 -20601.414} C_VEL
LIN {X 0,Y 211.572,Z 615.464,A -85,B 0,C 180,E1 -20604.281,E2 -20604.281} C_VEL
LIN {X 0,Y 211.573,Z 617.195,A -85,B 0,C 180,E1 -20606.191,E2 -20606.191} C_VEL
LIN {X 0,Y 211.675,Z 618.51,A -85,B 0,C 180,E1 -20608.097,E2 -20608.097} C_VEL
LIN {X 0,Y 211.741,Z 619.417,A -85,B 0,C 180,E1 -20610,E2 -20610} C_VEL
LIN {X 0,Y 211.644,Z 619.903,A -85,B 0,C 180,E1 -20611.903,E2 -20611.903} C_VEL
LIN {X 0,Y 211.498,Z 619.617,A -85,B 0,C 180,E1 -20615.721,E2 -20615.721} C_VEL
LIN {X 0,Y 212,Z 617.797,A -85,B 0,C 180,E1 -20619.541,E2 -20619.541} C_VEL
LIN {X 0,Y 212.517,Z 616.249,A -85,B 0,C 180,E1 -20621.444,E2 -20621.444} C_VEL
LIN {X 0,Y 213.661,Z 613.158,A -85,B 0,C 180,E1 -20624.282,E2 -20624.282} C_VEL
LIN {X 0,Y 215.464,Z 609.038,A -85,B 0,C 180,E1 -20627.071,E2 -20627.071} C_VEL
LIN {X 0,Y 218.111,Z 602.758,A -85,B 0,C 180,E1 -20630.266,E2 -20630.266} C_VEL
LIN {X 0,Y 220.738,Z 595.951,A -85,B 0,C 180,E1 -20632.955,E2 -20632.955} C_VEL
LIN {X 0,Y 223.988,Z 587.523,A -85,B 0,C 180,E1 -20635.558,E2 -20635.558} C_VEL
LIN {X 0,Y 227.243,Z 578.865,A -85,B 0,C 180,E1 -20637.639,E2 -20637.639} C_VEL
LIN {X 0,Y 230.703,Z 568.234,A -85,B 0,C 180,E1 -20639.671,E2 -20639.671} C_VEL
LIN {X 0,Y 233.781,Z 557.689,A -85,B 0,C 180,E1 -20641.236,E2 -20641.236} C_VEL
LIN {X 0,Y 236.567,Z 545.986,A -85,B 0,C 180,E1 -20642.578,E2 -20642.578} C_VEL
LIN {X 0,Y 238.958,Z 533.839,A -85,B 0,C 180,E1 -20643.592,E2 -20643.592} C_VEL
LIN {X 0,Y 240.809,Z 520.614,A -85,B 0,C 180,E1 -20644.369,E2 -20644.369} C_VEL
LIN {X 0,Y 241.883,Z 506.807,A -85,B 0,C 180,E1 -20644.857,E2 -20644.857} C_VEL
LIN {X 0,Y 243.625,Z 468.719,A -85,B 0,C 180,E1 -20645.95,E2 -20645.95} C_VEL
LIN {X 0,Y 241.261,Z 451.897,A -85,B 0,C 180,E1 -20647.059,E2 -20647.059} C_VEL
LIN {X 0,Y 234.765,Z 437.262,A -85,B 0,C 180,E1 -20649.027,E2 -20649.027} C_VEL
LIN {X 0,Y 228.432,Z 424.874,A -85,B 0,C 180,E1 -20651.04,E2 -20651.04} C_VEL
LIN {X 0,Y 222.702,Z 414.906,A -85,B 0,C 180,E1 -20652.973,E2 -20652.973} C_VEL
LIN {X 0,Y 219.702,Z 409.901,A -85,B 0,C 180,E1 -20654.045,E2 -20654.045} C_VEL
LIN {X 0,Y 217.102,Z 405.78,A -85,B 0,C 180,E1 -20655.007,E2 -20655.007} C_VEL
LIN {X 0,Y 216.703,Z 404.87,A -85,B 0,C 180,E1 -20655.2,E2 -20655.2} C_VEL
LIN {X 0,Y 214.906,Z 398.741,A -85,B 0,C 180,E1 -20659.152,E2 -20659.152} C_VEL
LIN {X 0,Y 213.759,Z 394.854,A -85,B 0,C 180,E1 -20661.942,E2 -20661.942} C_VEL
LIN {X 0,Y 213.766,Z 394.855,A -85,B 0,C 180,E1 -20666.02,E2 -20666.02} C_VEL
LIN {X 0,Y 213.777,Z 394.851,A -85,B 0,C 180,E1 -20670.454,E2 -20670.454} C_VEL
LIN {X 0,Y 213.797,Z 394.817,A -85,B 0,C 180,E1 -20674.701,E2 -20674.701} C_VEL
LIN {X 0,Y 213.809,Z 394.852,A -85,B 0,C 180,E1 -20678.803,E2 -20678.803} C_VEL
LIN {X 0,Y 213.939,Z 394.836,A -85,B 0,C 180,E1 -20682.804,E2 -20682.804} C_VEL
LIN {X 0,Y 213.975,Z 394.83,A -85,B 0,C 180,E1 -20686.708,E2 -20686.708} C_VEL
LIN {X 0,Y 214.163,Z 394.801,A -85,B 0,C 180,E1 -20690.557,E2 -20690.557} C_VEL
LIN {X 0,Y 214.236,Z 394.797,A -85,B 0,C 180,E1 -20692.46,E2 -20692.46} C_VEL
LIN {X 0,Y 214.442,Z 394.763,A -85,B 0,C 180,E1 -20698.122,E2 -20698.122} C_VEL
LIN {X 0,Y 214.55,Z 394.754,A -85,B 0,C 180,E1 -20700,E2 -20700} C_VEL
LIN {X 0,Y 214.441,Z 394.772,A -85,B 0,C 180,E1 -20701.879,E2 -20701.879} C_VEL
LIN {X 0,Y 214.194,Z 394.794,A -85,B 0,C 180,E1 -20707.542,E2 -20707.542} C_VEL
LIN {X 0,Y 213.995,Z 394.825,A -85,B 0,C 180,E1 -20711.365,E2 -20711.365} C_VEL
LIN {X 0,Y 213.926,Z 394.837,A -85,B 0,C 180,E1 -20715.238,E2 -20715.238} C_VEL
LIN {X 0,Y 213.865,Z 394.845,A -85,B 0,C 180,E1 -20719.186,E2 -20719.186} C_VEL
LIN {X 0,Y 213.845,Z 394.848,A -85,B 0,C 180,E1 -20723.228,E2 -20723.228} C_VEL
LIN {X 0,Y 213.827,Z 394.82,A -85,B 0,C 180,E1 -20727.451,E2 -20727.451} C_VEL
LIN {X 0,Y 213.778,Z 394.851,A -85,B 0,C 180,E1 -20731.737,E2 -20731.737} C_VEL
LIN {X 0,Y 213.768,Z 394.861,A -85,B 0,C 180,E1 -20735.091,E2 -20735.091} C_VEL
LIN {X 0,Y 214.565,Z 397.394,A -85,B 0,C 180,E1 -20735.477,E2 -20735.477} C_VEL
LIN {X 0,Y 216.463,Z 399.61,A -85,B 0,C 180,E1 -20736.18,E2 -20736.18} C_VEL
LIN {X 0,Y 217.476,Z 400.692,A -85,B 0,C 180,E1 -20736.542,E2 -20736.542} C_VEL
LIN {X 0,Y 219.571,Z 403.89,A -85,B 0,C 180,E1 -20737.318,E2 -20737.318} C_VEL
LIN {X 0,Y 220.761,Z 405.214,A -85,B 0,C 180,E1 -20737.722,E2 -20737.722} C_VEL
LIN {X 0,Y 227.552,Z 415.166,A -85,B 0,C 180,E1 -20740.002,E2 -20740.002} C_VEL
LIN {X 0,Y 235.423,Z 427.587,A -85,B 0,C 180,E1 -20742.415,E2 -20742.415} C_VEL
LIN {X 0,Y 240.69,Z 437.636,A -85,B 0,C 180,E1 -20743.958,E2 -20743.958} C_VEL
LIN {X 0,Y 244.65,Z 446.411,A -85,B 0,C 180,E1 -20745.098,E2 -20745.098} C_VEL
LIN {X 0,Y 242.114,Z 497.35,A -85,B 0,C 180,E1 -20746.577,E2 -20746.577} C_VEL
LIN {X 0,Y 240.778,Z 510.278,A -85,B 0,C 180,E1 -20747.238,E2 -20747.238} C_VEL
LIN {X 0,Y 238.856,Z 523.433,A -85,B 0,C 180,E1 -20748.264,E2 -20748.264} C_VEL
LIN {X 0,Y 236.382,Z 534.735,A -85,B 0,C 180,E1 -20749.431,E2 -20749.431} C_VEL
LIN {X 0,Y 233.586,Z 546.17,A -85,B 0,C 180,E1 -20751.032,E2 -20751.032} C_VEL
LIN {X 0,Y 230.524,Z 556.968,A -85,B 0,C 180,E1 -20752.979,E2 -20752.979} C_VEL
LIN {X 0,Y 227.267,Z 566.32,A -85,B 0,C 180,E1 -20755.105,E2 -20755.105} C_VEL
LIN {X 0,Y 223.856,Z 575.359,A -85,B 0,C 180,E1 -20757.744,E2 -20757.744} C_VEL
LIN {X 0,Y 220.872,Z 582.581,A -85,B 0,C 180,E1 -20760.45,E2 -20760.45} C_VEL
LIN {X 0,Y 218.285,Z 588.284,A -85,B 0,C 180,E1 -20763.209,E2 -20763.209} C_VEL
LIN {X 0,Y 216.019,Z 592.877,A -85,B 0,C 180,E1 -20766.117,E2 -20766.117} C_VEL
LIN {X 0,Y 214.415,Z 596.083,A -85,B 0,C 180,E1 -20768.866,E2 -20768.866} C_VEL
LIN {X 0,Y 213.561,Z 597.726,A -85,B 0,C 180,E1 -20770.787,E2 -20770.787} C_VEL
LIN {X 0,Y 212.665,Z 599.294,A -85,B 0,C 180,E1 -20773.413,E2 -20773.413} C_VEL
LIN {X 0,Y 211.878,Z 600.156,A -85,B 0,C 180,E1 -20776.574,E2 -20776.574} C_VEL
LIN {X 0,Y 211.509,Z 599.751,A -85,B 0,C 180,E1 -20780.437,E2 -20780.437} C_VEL
LIN {X 0,Y 211.555,Z 598.949,A -85,B 0,C 180,E1 -20782.364,E2 -20782.364} C_VEL
LIN {X 0,Y 211.803,Z 597.511,A -85,B 0,C 180,E1 -20784.543,E2 -20784.543} C_VEL
LIN {X 0,Y 212.147,Z 594.053,A -85,B 0,C 180,E1 -20788.102,E2 -20788.102} C_VEL
LIN {X 0,Y 212.866,Z 590.102,A -85,B 0,C 180,E1 -20790.946,E2 -20790.946} C_VEL
LIN {X 0,Y 213.863,Z 585.024,A -85,B 0,C 180,E1 -20793.768,E2 -20793.768} C_VEL
LIN {X 0,Y 215.279,Z 578.627,A -85,B 0,C 180,E1 -20796.561,E2 -20796.561} C_VEL
LIN {X 0,Y 217.033,Z 570.663,A -85,B 0,C 180,E1 -20799.318,E2 -20799.318} C_VEL
LIN {X 0,Y 218.826,Z 562.542,A -85,B 0,C 180,E1 -20801.579,E2 -20801.579} C_VEL
LIN {X 0,Y 220.967,Z 552.628,A -85,B 0,C 180,E1 -20803.8,E2 -20803.8} C_VEL
LIN {X 0,Y 223.04,Z 541.437,A -85,B 0,C 180,E1 -20805.769,E2 -20805.769} C_VEL
LIN {X 0,Y 224.706,Z 530.505,A -85,B 0,C 180,E1 -20807.285,E2 -20807.285} C_VEL
LIN {X 0,Y 226.25,Z 518.398,A -85,B 0,C 180,E1 -20808.565,E2 -20808.565} C_VEL
LIN {X 0,Y 227.42,Z 505.74,A -85,B 0,C 180,E1 -20809.52,E2 -20809.52} C_VEL
LIN {X 0,Y 228.149,Z 493.362,A -85,B 0,C 180,E1 -20810.122,E2 -20810.122} C_VEL
LIN {X 0,Y 230.46,Z 431.247,A -85,B 0,C 180,E1 -20811.991,E2 -20811.991} C_VEL
LIN {X 0,Y 225.772,Z 418.956,A -85,B 0,C 180,E1 -20813.051,E2 -20813.051} C_VEL
LIN {X 0,Y 218.648,Z 404.589,A -85,B 0,C 180,E1 -20814.605,E2 -20814.605} C_VEL
LIN {X 0,Y 214.005,Z 395.687,A -85,B 0,C 180,E1 -20815.669,E2 -20815.669} C_VEL
LIN {X 0,Y 213.866,Z 394.833,A -85,B 0,C 180,E1 -20815.812,E2 -20815.812} C_VEL
LIN {X 0,Y 213.797,Z 394.853,A -85,B 0,C 180,E1 -20821.274,E2 -20821.274} C_VEL
LIN {X 0,Y 213.746,Z 394.86,A -85,B 0,C 180,E1 -20826.287,E2 -20826.287} C_VEL
LIN {X 0,Y 213.718,Z 394.851,A -85,B 0,C 180,E1 -20831.123,E2 -20831.123} C_VEL
LIN {X 0,Y 213.748,Z 394.857,A -85,B 0,C 180,E1 -20833.667,E2 -20833.667} C_VEL
LIN {X 0,Y 213.812,Z 394.839,A -85,B 0,C 180,E1 -20836.347,E2 -20836.347} C_VEL
LIN {X 0,Y 213.797,Z 394.847,A -85,B 0,C 180,E1 -20839.117,E2 -20839.117} C_VEL
LIN {X 0,Y 213.753,Z 394.848,A -85,B 0,C 180,E1 -20843.713,E2 -20843.713} C_VEL
LIN {X 0,Y 213.768,Z 394.854,A -85,B 0,C 180,E1 -20848.262,E2 -20848.262} C_VEL
LIN {X 0,Y 213.824,Z 394.838,A -85,B 0,C 180,E1 -20852.602,E2 -20852.602} C_VEL
LIN {X 0,Y 213.86,Z 394.841,A -85,B 0,C 180,E1 -20856.946,E2 -20856.946} C_VEL
LIN {X 0,Y 213.93,Z 394.825,A -85,B 0,C 180,E1 -20862.304,E2 -20862.304} C_VEL
LIN {X 0,Y 213.949,Z 394.825,A -85,B 0,C 180,E1 -20866.706,E2 -20866.706} C_VEL
LIN {X 0,Y 214.163,Z 394.805,A -85,B 0,C 180,E1 -20870.556,E2 -20870.556} C_VEL
LIN {X 0,Y 214.223,Z 394.79,A -85,B 0,C 180,E1 -20872.459,E2 -20872.459} C_VEL
LIN {X 0,Y 214.441,Z 394.766,A -85,B 0,C 180,E1 -20878.121,E2 -20878.121} C_VEL
LIN {X 0,Y 214.55,Z 394.759,A -85,B 0,C 180,E1 -20880,E2 -20880} C_VEL
LIN {X 0,Y 214.442,Z 394.771,A -85,B 0,C 180,E1 -20881.878,E2 -20881.878} C_VEL
LIN {X 0,Y 214.223,Z 394.798,A -85,B 0,C 180,E1 -20887.54,E2 -20887.54} C_VEL
LIN {X 0,Y 214.04,Z 394.822,A -85,B 0,C 180,E1 -20891.362,E2 -20891.362} C_VEL
LIN {X 0,Y 213.928,Z 394.835,A -85,B 0,C 180,E1 -20895.237,E2 -20895.237} C_VEL
LIN {X 0,Y 213.872,Z 394.838,A -85,B 0,C 180,E1 -20899.184,E2 -20899.184} C_VEL
LIN {X 0,Y 213.852,Z 394.844,A -85,B 0,C 180,E1 -20903.226,E2 -20903.226} C_VEL
LIN {X 0,Y 213.825,Z 394.85,A -85,B 0,C 180,E1 -20907.45,E2 -20907.45} C_VEL
LIN {X 0,Y 213.766,Z 394.859,A -85,B 0,C 180,E1 -20911.737,E2 -20911.737} C_VEL
LIN {X 0,Y 213.751,Z 394.86,A -85,B 0,C 180,E1 -20916.287,E2 -20916.287} C_VEL
LIN {X 0,Y 213.791,Z 394.854,A -85,B 0,C 180,E1 -20921.106,E2 -20921.106} C_VEL
LIN {X 0,Y 213.806,Z 394.854,A -85,B 0,C 180,E1 -20923.685,E2 -20923.685} C_VEL
LIN {X 0,Y 213.714,Z 394.861,A -85,B 0,C 180,E1 -20928.228,E2 -20928.228} C_VEL
LIN {X 0,Y 213.173,Z 395.462,A -85,B 0,C 180,E1 -20929.262,E2 -20929.262} C_VEL
LIN {X 0,Y 211.919,Z 396.921,A -85,B 0,C 180,E1 -20930.214,E2 -20930.214} C_VEL
LIN {X 0,Y 208.918,Z 401.936,A -85,B 0,C 180,E1 -20932.303,E2 -20932.303} C_VEL
LIN {X 0,Y 208.774,Z 404.13,A -85,B 0,C 180,E1 -20933.254,E2 -20933.254} C_VEL
LIN {X 0,Y 209.319,Z 406.529,A -85,B 0,C 180,E1 -20934.34,E2 -20934.34} C_VEL
LIN {X 0,Y 216.916,Z 424.709,A -85,B 0,C 180,E1 -20936.244,E2 -20936.244} C_VEL
LIN {X 0,Y 219.583,Z 432.267,A -85,B 0,C 180,E1 -20936.917,E2 -20936.917} C_VEL
LIN {X 0,Y 223.121,Z 465.506,A -85,B 0,C 180,E1 -20938.608,E2 -20938.608} C_VEL
LIN {X 0,Y 221.137,Z 515.178,A -85,B 0,C 180,E1 -20940.161,E2 -20940.161} C_VEL
LIN {X 0,Y 220.051,Z 528.591,A -85,B 0,C 180,E1 -20940.919,E2 -20940.919} C_VEL
LIN {X 0,Y 218.483,Z 540.82,A -85,B 0,C 180,E1 -20941.937,E2 -20941.937} C_VEL
LIN {X 0,Y 216.662,Z 552.339,A -85,B 0,C 180,E1 -20943.252,E2 -20943.252} C_VEL
LIN {X 0,Y 214.338,Z 564.141,A -85,B 0,C 180,E1 -20945.029,E2 -20945.029} C_VEL
LIN {X 0,Y 212.107,Z 574.747,A -85,B 0,C 180,E1 -20947.088,E2 -20947.088} C_VEL
LIN {X 0,Y 210.011,Z 584.341,A -85,B 0,C 180,E1 -20949.441,E2 -20949.441} C_VEL
LIN {X 0,Y 208.436,Z 592.131,A -85,B 0,C 180,E1 -20951.827,E2 -20951.827} C_VEL
LIN {X 0,Y 206.76,Z 599.765,A -85,B 0,C 180,E1 -20954.727,E2 -20954.727} C_VEL
LIN {X 0,Y 205.381,Z 606.813,A -85,B 0,C 180,E1 -20958.152,E2 -20958.152} C_VEL
LIN {X 0,Y 204.781,Z 611.47,A -85,B 0,C 180,E1 -20961.116,E2 -20961.116} C_VEL
LIN {X 0,Y 204.496,Z 614.997,A -85,B 0,C 180,E1 -20964.082,E2 -20964.082} C_VEL
LIN {X 0,Y 204.478,Z 616.764,A -85,B 0,C 180,E1 -20966.058,E2 -20966.058} C_VEL
LIN {X 0,Y 204.585,Z 618.102,A -85,B 0,C 180,E1 -20968.031,E2 -20968.031} C_VEL
LIN {X 0,Y 204.674,Z 619.032,A -85,B 0,C 180,E1 -20970,E2 -20970} C_VEL
LIN {X 0,Y 204.553,Z 619.549,A -85,B 0,C 180,E1 -20971.969,E2 -20971.969} C_VEL
LIN {X 0,Y 204.438,Z 619.574,A -85,B 0,C 180,E1 -20974.487,E2 -20974.487} C_VEL
LIN {X 0,Y 204.593,Z 618.618,A -85,B 0,C 180,E1 -20977.897,E2 -20977.897} C_VEL
LIN {X 0,Y 204.964,Z 617.54,A -85,B 0,C 180,E1 -20979.872,E2 -20979.872} C_VEL
LIN {X 0,Y 205.521,Z 616.031,A -85,B 0,C 180,E1 -20981.839,E2 -20981.839} C_VEL
LIN {X 0,Y 206.748,Z 612.985,A -85,B 0,C 180,E1 -20984.77,E2 -20984.77} C_VEL
LIN {X 0,Y 208.66,Z 608.913,A -85,B 0,C 180,E1 -20987.645,E2 -20987.645} C_VEL
LIN {X 0,Y 211.445,Z 602.688,A -85,B 0,C 180,E1 -20990.934,E2 -20990.934} C_VEL
LIN {X 0,Y 214.19,Z 595.942,A -85,B 0,C 180,E1 -20993.699,E2 -20993.699} C_VEL
LIN {X 0,Y 217.612,Z 587.606,A -85,B 0,C 180,E1 -20996.363,E2 -20996.363} C_VEL
LIN {X 0,Y 220.974,Z 579.051,A -85,B 0,C 180,E1 -20998.493,E2 -20998.493} C_VEL
LIN {X 0,Y 224.579,Z 568.529,A -85,B 0,C 180,E1 -21000.565,E2 -21000.565} C_VEL
LIN {X 0,Y 227.775,Z 558.12,A -85,B 0,C 180,E1 -21002.157,E2 -21002.157} C_VEL
LIN {X 0,Y 230.644,Z 546.705,A -85,B 0,C 180,E1 -21003.523,E2 -21003.523} C_VEL
LIN {X 0,Y 233.34,Z 533.613,A -85,B 0,C 180,E1 -21004.645,E2 -21004.645} C_VEL
LIN {X 0,Y 235.229,Z 520.399,A -85,B 0,C 180,E1 -21005.439,E2 -21005.439} C_VEL
LIN {X 0,Y 236.35,Z 507.109,A -85,B 0,C 180,E1 -21005.915,E2 -21005.915} C_VEL
LIN {X 0,Y 238.148,Z 469.839,A -85,B 0,C 180,E1 -21007,E2 -21007} C_VEL
LIN {X 0,Y 236.03,Z 454.683,A -85,B 0,C 180,E1 -21008.045,E2 -21008.045} C_VEL
LIN {X 0,Y 230.052,Z 441.061,A -85,B 0,C 180,E1 -21009.953,E2 -21009.953} C_VEL
LIN {X 0,Y 224.371,Z 429.715,A -85,B 0,C 180,E1 -21011.857,E2 -21011.857} C_VEL
LIN {X 0,Y 218.343,Z 419.13,A -85,B 0,C 180,E1 -21013.994,E2 -21013.994} C_VEL
LIN {X 0,Y 215.594,Z 414.559,A -85,B 0,C 180,E1 -21015.028,E2 -21015.028} C_VEL
LIN {X 0,Y 212.484,Z 409.513,A -85,B 0,C 180,E1 -21016.253,E2 -21016.253} C_VEL
LIN {X 0,Y 209.67,Z 405.122,A -85,B 0,C 180,E1 -21017.413,E2 -21017.413} C_VEL
LIN {X 0,Y 209.339,Z 404.325,A -85,B 0,C 180,E1 -21017.61,E2 -21017.61} C_VEL
LIN {X 0,Y 207.866,Z 399.418,A -85,B 0,C 180,E1 -21021.043,E2 -21021.043} C_VEL
LIN {X 0,Y 206.711,Z 395.732,A -85,B 0,C 180,E1 -21023.943,E2 -21023.943} C_VEL
LIN {X 0,Y 206.725,Z 395.735,A -85,B 0,C 180,E1 -21028.201,E2 -21028.201} C_VEL
LIN {X 0,Y 206.763,Z 395.725,A -85,B 0,C 180,E1 -21032.096,E2 -21032.096} C_VEL
LIN {X 0,Y 206.781,Z 395.698,A -85,B 0,C 180,E1 -21036.584,E2 -21036.584} C_VEL
LIN {X 0,Y 206.869,Z 395.713,A -85,B 0,C 180,E1 -21042.197,E2 -21042.197} C_VEL
LIN {X 0,Y 206.908,Z 395.706,A -85,B 0,C 180,E1 -21046.246,E2 -21046.246} C_VEL
LIN {X 0,Y 207.101,Z 395.678,A -85,B 0,C 180,E1 -21050.231,E2 -21050.231} C_VEL
LIN {X 0,Y 207.174,Z 395.679,A -85,B 0,C 180,E1 -21052.202,E2 -21052.202} C_VEL
LIN {X 0,Y 207.379,Z 395.643,A -85,B 0,C 180,E1 -21058.058,E2 -21058.058} C_VEL
LIN {X 0,Y 207.514,Z 395.63,A -85,B 0,C 180,E1 -21060,E2 -21060} C_VEL
LIN {X 0,Y 207.378,Z 395.65,A -85,B 0,C 180,E1 -21061.943,E2 -21061.943} C_VEL
LIN {X 0,Y 207.137,Z 395.672,A -85,B 0,C 180,E1 -21067.801,E2 -21067.801} C_VEL
LIN {X 0,Y 206.919,Z 395.703,A -85,B 0,C 180,E1 -21071.759,E2 -21071.759} C_VEL
LIN {X 0,Y 206.86,Z 395.713,A -85,B 0,C 180,E1 -21075.772,E2 -21075.772} C_VEL
LIN {X 0,Y 206.796,Z 395.721,A -85,B 0,C 180,E1 -21079.869,E2 -21079.869} C_VEL
LIN {X 0,Y 206.761,Z 395.717,A -85,B 0,C 180,E1 -21084.073,E2 -21084.073} C_VEL
LIN {X 0,Y 206.742,Z 395.713,A -85,B 0,C 180,E1 -21088.42,E2 -21088.42} C_VEL
LIN {X 0,Y 206.69,Z 395.741,A -85,B 0,C 180,E1 -21092.71,E2 -21092.71} C_VEL
LIN {X 0,Y 207.55,Z 398.319,A -85,B 0,C 180,E1 -21093.168,E2 -21093.168} C_VEL
LIN {X 0,Y 209.628,Z 400.62,A -85,B 0,C 180,E1 -21094.02,E2 -21094.02} C_VEL
LIN {X 0,Y 210.387,Z 401.294,A -85,B 0,C 180,E1 -21094.314,E2 -21094.314} C_VEL
LIN {X 0,Y 212.292,Z 404.442,A -85,B 0,C 180,E1 -21095.11,E2 -21095.11} C_VEL
LIN {X 0,Y 214.09,Z 406.394,A -85,B 0,C 180,E1 -21095.785,E2 -21095.785} C_VEL
LIN {X 0,Y 216.717,Z 410.073,A -85,B 0,C 180,E1 -21096.776,E2 -21096.776} C_VEL
LIN {X 0,Y 223.152,Z 419.399,A -85,B 0,C 180,E1 -21099.042,E2 -21099.042} C_VEL
LIN {X 0,Y 231.967,Z 433.681,A -85,B 0,C 180,E1 -21101.874,E2 -21101.874} C_VEL
LIN {X 0,Y 237.804,Z 445.656,A -85,B 0,C 180,E1 -21103.665,E2 -21103.665} C_VEL
LIN {X 0,Y 239.218,Z 448.771,A -85,B 0,C 180,E1 -21104.086,E2 -21104.086} C_VEL
LIN {X 0,Y 236.586,Z 497.905,A -85,B 0,C 180,E1 -21105.525,E2 -21105.525} C_VEL
LIN {X 0,Y 235.143,Z 511.102,A -85,B 0,C 180,E1 -21106.216,E2 -21106.216} C_VEL
LIN {X 0,Y 233.307,Z 523.269,A -85,B 0,C 180,E1 -21107.184,E2 -21107.184} C_VEL
LIN {X 0,Y 230.524,Z 535.519,A -85,B 0,C 180,E1 -21108.465,E2 -21108.465} C_VEL
LIN {X 0,Y 227.605,Z 546.893,A -85,B 0,C 180,E1 -21110.097,E2 -21110.097} C_VEL
LIN {X 0,Y 224.419,Z 557.594,A -85,B 0,C 180,E1 -21112.079,E2 -21112.079} C_VEL
LIN {X 0,Y 221.359,Z 566.058,A -85,B 0,C 180,E1 -21114.031,E2 -21114.031} C_VEL
LIN {X 0,Y 217.725,Z 575.195,A -85,B 0,C 180,E1 -21116.72,E2 -21116.72} C_VEL
LIN {X 0,Y 214.583,Z 582.516,A -85,B 0,C 180,E1 -21119.493,E2 -21119.493} C_VEL
LIN {X 0,Y 211.826,Z 588.32,A -85,B 0,C 180,E1 -21122.323,E2 -21122.323} C_VEL
LIN {X 0,Y 209.861,Z 592.151,A -85,B 0,C 180,E1 -21124.718,E2 -21124.718} C_VEL
LIN {X 0,Y 207.652,Z 596.256,A -85,B 0,C 180,E1 -21128.143,E2 -21128.143} C_VEL
LIN {X 0,Y 206.706,Z 597.931,A -85,B 0,C 180,E1 -21130.124,E2 -21130.124} C_VEL
LIN {X 0,Y 205.641,Z 599.671,A -85,B 0,C 180,E1 -21133.125,E2 -21133.125} C_VEL
LIN {X 0,Y 204.881,Z 600.479,A -85,B 0,C 180,E1 -21136.107,E2 -21136.107} C_VEL
LIN {X 0,Y 204.437,Z 600.132,A -85,B 0,C 180,E1 -21140.103,E2 -21140.103} C_VEL
LIN {X 0,Y 204.442,Z 599.378,A -85,B 0,C 180,E1 -21142.097,E2 -21142.097} C_VEL
LIN {X 0,Y 204.712,Z 597.771,A -85,B 0,C 180,E1 -21144.635,E2 -21144.635} C_VEL
LIN {X 0,Y 205.057,Z 594.581,A -85,B 0,C 180,E1 -21148.036,E2 -21148.036} C_VEL
LIN {X 0,Y 205.783,Z 590.694,A -85,B 0,C 180,E1 -21150.978,E2 -21150.978} C_VEL
LIN {X 0,Y 206.795,Z 585.691,A -85,B 0,C 180,E1 -21153.897,E2 -21153.897} C_VEL
LIN {X 0,Y 208.229,Z 579.405,A -85,B 0,C 180,E1 -21156.784,E2 -21156.784} C_VEL
LIN {X 0,Y 210.052,Z 571.538,A -85,B 0,C 180,E1 -21159.63,E2 -21159.63} C_VEL
LIN {X 0,Y 212.319,Z 561.75,A -85,B 0,C 180,E1 -21162.424,E2 -21162.424} C_VEL
LIN {X 0,Y 214.566,Z 551.514,A -85,B 0,C 180,E1 -21164.705,E2 -21164.705} C_VEL
LIN {X 0,Y 216.777,Z 539.97,A -85,B 0,C 180,E1 -21166.722,E2 -21166.722} C_VEL
LIN {X 0,Y 218.502,Z 528.607,A -85,B 0,C 180,E1 -21168.276,E2 -21168.276} C_VEL
LIN {X 0,Y 220.01,Z 516.841,A -85,B 0,C 180,E1 -21169.476,E2 -21169.476} C_VEL
LIN {X 0,Y 221.207,Z 503.3,A -85,B 0,C 180,E1 -21170.455,E2 -21170.455} C_VEL
LIN {X 0,Y 221.905,Z 490.862,A -85,B 0,C 180,E1 -21171.007,E2 -21171.007} C_VEL
LIN {X 0,Y 224.097,Z 432.689,A -85,B 0,C 180,E1 -21172.791,E2 -21172.791} C_VEL
LIN {X 0,Y 219.868,Z 421.77,A -85,B 0,C 180,E1 -21173.787,E2 -21173.787} C_VEL
LIN {X 0,Y 211.843,Z 405.629,A -85,B 0,C 180,E1 -21175.635,E2 -21175.635} C_VEL
LIN {X 0,Y 207.902,Z 398.701,A -85,B 0,C 180,E1 -21176.57,E2 -21176.57} C_VEL
LIN {X 0,Y 206.864,Z 396.121,A -85,B 0,C 180,E1 -21176.854,E2 -21176.854} C_VEL
LIN {X 0,Y 206.796,Z 395.721,A -85,B 0,C 180,E1 -21176.934,E2 -21176.934} C_VEL
LIN {X 0,Y 206.729,Z 395.734,A -85,B 0,C 180,E1 -21181.797,E2 -21181.797} C_VEL
LIN {X 0,Y 206.7,Z 395.737,A -85,B 0,C 180,E1 -21185.31,E2 -21185.31} C_VEL
LIN {X 0,Y 206.664,Z 395.732,A -85,B 0,C 180,E1 -21190.249,E2 -21190.249} C_VEL
LIN {X 0,Y 206.708,Z 395.732,A -85,B 0,C 180,E1 -21195.559,E2 -21195.559} C_VEL
LIN {X 0,Y 206.727,Z 395.729,A -85,B 0,C 180,E1 -21199.763,E2 -21199.763} C_VEL
LIN {X 0,Y 206.725,Z 395.731,A -85,B 0,C 180,E1 -21202.269,E2 -21202.269} C_VEL
LIN {X 0,Y 206.704,Z 395.728,A -85,B 0,C 180,E1 -21207.042,E2 -21207.042} C_VEL
LIN {X 0,Y 206.762,Z 395.721,A -85,B 0,C 180,E1 -21212.097,E2 -21212.097} C_VEL
LIN {X 0,Y 206.79,Z 395.717,A -85,B 0,C 180,E1 -21216.578,E2 -21216.578} C_VEL
LIN {X 0,Y 206.875,Z 395.704,A -85,B 0,C 180,E1 -21222.196,E2 -21222.196} C_VEL
LIN {X 0,Y 206.891,Z 395.698,A -85,B 0,C 180,E1 -21226.243,E2 -21226.243} C_VEL
LIN {X 0,Y 207.102,Z 395.687,A -85,B 0,C 180,E1 -21230.231,E2 -21230.231} C_VEL
LIN {X 0,Y 207.164,Z 395.67,A -85,B 0,C 180,E1 -21232.2,E2 -21232.2} C_VEL
LIN {X 0,Y 207.378,Z 395.645,A -85,B 0,C 180,E1 -21238.057,E2 -21238.057} C_VEL
LIN {X 0,Y 207.514,Z 395.636,A -85,B 0,C 180,E1 -21240,E2 -21240} C_VEL
LIN {X 0,Y 207.082,Z 395.684,A -85,B 0,C 180,E1 -21243.892,E2 -21243.892} C_VEL
LIN {X 0,Y 207.163,Z 395.676,A -85,B 0,C 180,E1 -21247.799,E2 -21247.799} C_VEL
LIN {X 0,Y 206.977,Z 395.704,A -85,B 0,C 180,E1 -21251.755,E2 -21251.755} C_VEL
LIN {X 0,Y 206.862,Z 395.717,A -85,B 0,C 180,E1 -21255.771,E2 -21255.771} C_VEL
LIN {X 0,Y 206.809,Z 395.721,A -85,B 0,C 180,E1 -21259.866,E2 -21259.866} C_VEL
LIN {X 0,Y 206.764,Z 395.727,A -85,B 0,C 180,E1 -21264.072,E2 -21264.072} C_VEL
LIN {X 0,Y 206.733,Z 395.731,A -85,B 0,C 180,E1 -21268.42,E2 -21268.42} C_VEL
LIN {X 0,Y 206.702,Z 395.738,A -85,B 0,C 180,E1 -21272.957,E2 -21272.957} C_VEL
LIN {X 0,Y 206.722,Z 395.737,A -85,B 0,C 180,E1 -21277.73,E2 -21277.73} C_VEL
LIN {X 0,Y 206.721,Z 395.734,A -85,B 0,C 180,E1 -21281.589,E2 -21281.589} C_VEL
LIN {X 0,Y 206.693,Z 395.738,A -85,B 0,C 180,E1 -21285.564,E2 -21285.564} C_VEL
LIN {X 0,Y 206.74,Z 395.908,A -85,B 0,C 180,E1 -21289.177,E2 -21289.177} C_VEL
LIN {X 0,Y 208.774,Z 404.13,A -85,B 0,C 180,E1 -21293.254,E2 -21293.254} C_VEL
LIN {X 0,Y 209.037,Z 406.35,A -85,B 0,C 180,E1 -21293.885,E2 -21293.885} C_VEL
LIN {X 0,Y 209.043,Z 410.607,A -85,B 0,C 180,E1 -21294.389,E2 -21294.389} C_VEL
LIN {X 0,Y 208.902,Z 420.348,A -85,B 0,C 180,E1 -21294.814,E2 -21294.814} C_VEL
LIN {X 0,Y 209.823,Z 424.281,A -85,B 0,C 180,E1 -21295.122,E2 -21295.122} C_VEL
LIN {X 0,Y 213.528,Z 434.579,A -85,B 0,C 180,E1 -21296.103,E2 -21296.103} C_VEL
LIN {X 0,Y 216.777,Z 465.27,A -85,B 0,C 180,E1 -21297.732,E2 -21297.732} C_VEL
LIN {X 0,Y 214.813,Z 514.69,A -85,B 0,C 180,E1 -21299.325,E2 -21299.325} C_VEL
LIN {X 0,Y 213.77,Z 527.396,A -85,B 0,C 180,E1 -21300.046,E2 -21300.046} C_VEL
LIN {X 0,Y 212.049,Z 540.416,A -85,B 0,C 180,E1 -21301.142,E2 -21301.142} C_VEL
LIN {X 0,Y 210.003,Z 552.77,A -85,B 0,C 180,E1 -21302.603,E2 -21302.603} C_VEL
LIN {X 0,Y 207.608,Z 564.422,A -85,B 0,C 180,E1 -21304.431,E2 -21304.431} C_VEL
LIN {X 0,Y 205.301,Z 574.923,A -85,B 0,C 180,E1 -21306.55,E2 -21306.55} C_VEL
LIN {X 0,Y 203.087,Z 584.524,A -85,B 0,C 180,E1 -21309.014,E2 -21309.014} C_VEL
LIN {X 0,Y 201.293,Z 592.804,A -85,B 0,C 180,E1 -21311.686,E2 -21311.686} C_VEL
LIN {X 0,Y 199.612,Z 600.262,A -85,B 0,C 180,E1 -21314.689,E2 -21314.689} C_VEL
LIN {X 0,Y 198.384,Z 606.236,A -85,B 0,C 180,E1 -21317.728,E2 -21317.728} C_VEL
LIN {X 0,Y 197.723,Z 610.947,A -85,B 0,C 180,E1 -21320.796,E2 -21320.796} C_VEL
LIN {X 0,Y 197.41,Z 614.521,A -85,B 0,C 180,E1 -21323.869,E2 -21323.869} C_VEL
LIN {X 0,Y 197.413,Z 616.336,A -85,B 0,C 180,E1 -21325.917,E2 -21325.917} C_VEL
LIN {X 0,Y 197.497,Z 617.694,A -85,B 0,C 180,E1 -21327.961,E2 -21327.961} C_VEL
LIN {X 0,Y 197.608,Z 618.646,A -85,B 0,C 180,E1 -21330,E2 -21330} C_VEL
LIN {X 0,Y 197.464,Z 619.186,A -85,B 0,C 180,E1 -21332.04,E2 -21332.04} C_VEL
LIN {X 0,Y 197.338,Z 619.284,A -85,B 0,C 180,E1 -21334.298,E2 -21334.298} C_VEL
LIN {X 0,Y 197.528,Z 618.335,A -85,B 0,C 180,E1 -21338.182,E2 -21338.182} C_VEL
LIN {X 0,Y 197.946,Z 617.279,A -85,B 0,C 180,E1 -21340.225,E2 -21340.225} C_VEL
LIN {X 0,Y 198.545,Z 615.812,A -85,B 0,C 180,E1 -21342.262,E2 -21342.262} C_VEL
LIN {X 0,Y 199.86,Z 612.806,A -85,B 0,C 180,E1 -21345.291,E2 -21345.291} C_VEL
LIN {X 0,Y 201.865,Z 608.779,A -85,B 0,C 180,E1 -21348.26,E2 -21348.26} C_VEL
LIN {X 0,Y 204.787,Z 602.624,A -85,B 0,C 180,E1 -21351.649,E2 -21351.649} C_VEL
LIN {X 0,Y 207.682,Z 595.94,A -85,B 0,C 180,E1 -21354.49,E2 -21354.49} C_VEL
LIN {X 0,Y 211.282,Z 587.677,A -85,B 0,C 180,E1 -21357.217,E2 -21357.217} C_VEL
LIN {X 0,Y 214.775,Z 579.233,A -85,B 0,C 180,E1 -21359.395,E2 -21359.395} C_VEL
LIN {X 0,Y 218.518,Z 568.829,A -85,B 0,C 180,E1 -21361.508,E2 -21361.508} C_VEL
LIN {X 0,Y 222.194,Z 557.138,A -85,B 0,C 180,E1 -21363.337,E2 -21363.337} C_VEL
LIN {X 0,Y 225.272,Z 545.48,A -85,B 0,C 180,E1 -21364.705,E2 -21364.705} C_VEL
LIN {X 0,Y 227.803,Z 533.387,A -85,B 0,C 180,E1 -21365.749,E2 -21365.749} C_VEL
LIN {X 0,Y 229.747,Z 520.28,A -85,B 0,C 180,E1 -21366.549,E2 -21366.549} C_VEL
LIN {X 0,Y 230.918,Z 507.059,A -85,B 0,C 180,E1 -21367.035,E2 -21367.035} C_VEL
LIN {X 0,Y 232.758,Z 470.926,A -85,B 0,C 180,E1 -21368.1,E2 -21368.1} C_VEL
LIN {X 0,Y 230.98,Z 457.72,A -85,B 0,C 180,E1 -21369.039,E2 -21369.039} C_VEL
LIN {X 0,Y 224.982,Z 443.893,A -85,B 0,C 180,E1 -21371.069,E2 -21371.069} C_VEL
LIN {X 0,Y 219.343,Z 432.737,A -85,B 0,C 180,E1 -21373.066,E2 -21373.066} C_VEL
LIN {X 0,Y 214.128,Z 423.415,A -85,B 0,C 180,E1 -21375.032,E2 -21375.032} C_VEL
LIN {X 0,Y 211.617,Z 419.247,A -85,B 0,C 180,E1 -21376.028,E2 -21376.028} C_VEL
LIN {X 0,Y 208.881,Z 414.723,A -85,B 0,C 180,E1 -21377.164,E2 -21377.164} C_VEL
LIN {X 0,Y 205.436,Z 409.337,A -85,B 0,C 180,E1 -21378.664,E2 -21378.664} C_VEL
LIN {X 0,Y 202.451,Z 404.941,A -85,B 0,C 180,E1 -21380.033,E2 -21380.033} C_VEL
LIN {X 0,Y 201.904,Z 403.699,A -85,B 0,C 180,E1 -21380.385,E2 -21380.385} C_VEL
LIN {X 0,Y 200.263,Z 398.717,A -85,B 0,C 180,E1 -21384.351,E2 -21384.351} C_VEL
LIN {X 0,Y 199.644,Z 396.615,A -85,B 0,C 180,E1 -21386.251,E2 -21386.251} C_VEL
LIN {X 0,Y 199.671,Z 396.607,A -85,B 0,C 180,E1 -21390.478,E2 -21390.478} C_VEL
LIN {X 0,Y 199.669,Z 396.575,A -85,B 0,C 180,E1 -21395.015,E2 -21395.015} C_VEL
LIN {X 0,Y 199.696,Z 396.607,A -85,B 0,C 180,E1 -21399.395,E2 -21399.395} C_VEL
LIN {X 0,Y 199.799,Z 396.593,A -85,B 0,C 180,E1 -21403.657,E2 -21403.657} C_VEL
LIN {X 0,Y 199.909,Z 396.582,A -85,B 0,C 180,E1 -21407.823,E2 -21407.823} C_VEL
LIN {X 0,Y 200.115,Z 396.558,A -85,B 0,C 180,E1 -21411.925,E2 -21411.925} C_VEL
LIN {X 0,Y 200.318,Z 396.523,A -85,B 0,C 180,E1 -21417.99,E2 -21417.99} C_VEL
LIN {X 0,Y 200.478,Z 396.505,A -85,B 0,C 180,E1 -21420.001,E2 -21420.001} C_VEL
LIN {X 0,Y 200.023,Z 396.557,A -85,B 0,C 180,E1 -21424.03,E2 -21424.03} C_VEL
LIN {X 0,Y 200.085,Z 396.549,A -85,B 0,C 180,E1 -21428.077,E2 -21428.077} C_VEL
LIN {X 0,Y 199.87,Z 396.578,A -85,B 0,C 180,E1 -21432.18,E2 -21432.18} C_VEL
LIN {X 0,Y 199.8,Z 396.588,A -85,B 0,C 180,E1 -21436.345,E2 -21436.345} C_VEL
LIN {X 0,Y 199.821,Z 396.592,A -85,B 0,C 180,E1 -21438.455,E2 -21438.455} C_VEL
LIN {X 0,Y 199.734,Z 396.596,A -85,B 0,C 180,E1 -21443.818,E2 -21443.818} C_VEL
LIN {X 0,Y 199.711,Z 396.587,A -85,B 0,C 180,E1 -21448.388,E2 -21448.388} C_VEL
LIN {X 0,Y 199.662,Z 396.619,A -85,B 0,C 180,E1 -21450.033,E2 -21450.033} C_VEL
LIN {X 0,Y 200.519,Z 399.196,A -85,B 0,C 180,E1 -21450.546,E2 -21450.546} C_VEL
LIN {X 0,Y 202.597,Z 401.51,A -85,B 0,C 180,E1 -21451.51,E2 -21451.51} C_VEL
LIN {X 0,Y 203.556,Z 402.312,A -85,B 0,C 180,E1 -21451.925,E2 -21451.925} C_VEL
LIN {X 0,Y 205.587,Z 405.563,A -85,B 0,C 180,E1 -21452.867,E2 -21452.867} C_VEL
LIN {X 0,Y 207.333,Z 407.427,A -85,B 0,C 180,E1 -21453.596,E2 -21453.596} C_VEL
LIN {X 0,Y 209.945,Z 411.081,A -85,B 0,C 180,E1 -21454.687,E2 -21454.687} C_VEL
LIN {X 0,Y 216.485,Z 420.19,A -85,B 0,C 180,E1 -21457.204,E2 -21457.204} C_VEL
LIN {X 0,Y 223.678,Z 431.533,A -85,B 0,C 180,E1 -21459.733,E2 -21459.733} C_VEL
LIN {X 0,Y 228.996,Z 440.805,A -85,B 0,C 180,E1 -21461.472,E2 -21461.472} C_VEL
LIN {X 0,Y 233.793,Z 451.174,A -85,B 0,C 180,E1 -21463.013,E2 -21463.013} C_VEL
LIN {X 0,Y 231.129,Z 498.637,A -85,B 0,C 180,E1 -21464.432,E2 -21464.432} C_VEL
LIN {X 0,Y 229.628,Z 511.611,A -85,B 0,C 180,E1 -21465.123,E2 -21465.123} C_VEL
LIN {X 0,Y 227.616,Z 524.234,A -85,B 0,C 180,E1 -21466.15,E2 -21466.15} C_VEL
LIN {X 0,Y 224.736,Z 536.303,A -85,B 0,C 180,E1 -21467.449,E2 -21467.449} C_VEL
LIN {X 0,Y 221.91,Z 546.811,A -85,B 0,C 180,E1 -21468.978,E2 -21468.978} C_VEL
LIN {X 0,Y 218.746,Z 557.16,A -85,B 0,C 180,E1 -21470.912,E2 -21470.912} C_VEL
LIN {X 0,Y 215.548,Z 565.773,A -85,B 0,C 180,E1 -21472.902,E2 -21472.902} C_VEL
LIN {X 0,Y 212.322,Z 573.664,A -85,B 0,C 180,E1 -21475.182,E2 -21475.182} C_VEL
LIN {X 0,Y 208.898,Z 581.319,A -85,B 0,C 180,E1 -21478.003,E2 -21478.003} C_VEL
LIN {X 0,Y 205.415,Z 588.342,A -85,B 0,C 180,E1 -21481.381,E2 -21481.381} C_VEL
LIN {X 0,Y 203.108,Z 592.618,A -85,B 0,C 180,E1 -21484.115,E2 -21484.115} C_VEL
LIN {X 0,Y 200.931,Z 596.42,A -85,B 0,C 180,E1 -21487.372,E2 -21487.372} C_VEL
LIN {X 0,Y 199.905,Z 598.136,A -85,B 0,C 180,E1 -21489.417,E2 -21489.417} C_VEL
LIN {X 0,Y 198.42,Z 600.32,A -85,B 0,C 180,E1 -21493.54,E2 -21493.54} C_VEL
LIN {X 0,Y 197.905,Z 600.801,A -85,B 0,C 180,E1 -21495.607,E2 -21495.607} C_VEL
LIN {X 0,Y 197.345,Z 600.514,A -85,B 0,C 180,E1 -21499.743,E2 -21499.743} C_VEL
LIN {X 0,Y 197.358,Z 599.79,A -85,B 0,C 180,E1 -21501.811,E2 -21501.811} C_VEL
LIN {X 0,Y 197.627,Z 598.044,A -85,B 0,C 180,E1 -21504.714,E2 -21504.714} C_VEL
LIN {X 0,Y 198.127,Z 593.955,A -85,B 0,C 180,E1 -21508.984,E2 -21508.984} C_VEL
LIN {X 0,Y 198.988,Z 589.773,A -85,B 0,C 180,E1 -21512.024,E2 -21512.024} C_VEL
LIN {X 0,Y 200.364,Z 583.428,A -85,B 0,C 180,E1 -21515.535,E2 -21515.535} C_VEL
LIN {X 0,Y 202.087,Z 576.506,A -85,B 0,C 180,E1 -21518.499,E2 -21518.499} C_VEL
LIN {X 0,Y 204.239,Z 567.829,A -85,B 0,C 180,E1 -21521.412,E2 -21521.412} C_VEL
LIN {X 0,Y 206.306,Z 558.955,A -85,B 0,C 180,E1 -21523.795,E2 -21523.795} C_VEL
LIN {X 0,Y 208.473,Z 549.194,A -85,B 0,C 180,E1 -21525.897,E2 -21525.897} C_VEL
LIN {X 0,Y 210.579,Z 538.445,A -85,B 0,C 180,E1 -21527.73,E2 -21527.73} C_VEL
LIN {X 0,Y 212.351,Z 526.45,A -85,B 0,C 180,E1 -21529.327,E2 -21529.327} C_VEL
LIN {X 0,Y 213.98,Z 513.875,A -85,B 0,C 180,E1 -21530.549,E2 -21530.549} C_VEL
LIN {X 0,Y 215.013,Z 501.309,A -85,B 0,C 180,E1 -21531.404,E2 -21531.404} C_VEL
LIN {X 0,Y 215.745,Z 486.37,A -85,B 0,C 180,E1 -21531.991,E2 -21531.991} C_VEL
LIN {X 0,Y 217.788,Z 434.3,A -85,B 0,C 180,E1 -21533.627,E2 -21533.627} C_VEL
LIN {X 0,Y 214.16,Z 424.882,A -85,B 0,C 180,E1 -21534.527,E2 -21534.527} C_VEL
LIN {X 0,Y 205.955,Z 408.529,A -85,B 0,C 180,E1 -21536.511,E2 -21536.511} C_VEL
LIN {X 0,Y 201.136,Z 399.993,A -85,B 0,C 180,E1 -21537.728,E2 -21537.728} C_VEL
LIN {X 0,Y 199.899,Z 397.536,A -85,B 0,C 180,E1 -21538.064,E2 -21538.064} C_VEL
LIN {X 0,Y 199.716,Z 396.606,A -85,B 0,C 180,E1 -21538.188,E2 -21538.188} C_VEL
LIN {X 0,Y 199.681,Z 396.613,A -85,B 0,C 180,E1 -21542.358,E2 -21542.358} C_VEL
LIN {X 0,Y 199.625,Z 396.617,A -85,B 0,C 180,E1 -21546.762,E2 -21546.762} C_VEL
LIN {X 0,Y 199.611,Z 396.617,A -85,B 0,C 180,E1 -21549.326,E2 -21549.326} C_VEL
LIN {X 0,Y 199.632,Z 396.614,A -85,B 0,C 180,E1 -21554.755,E2 -21554.755} C_VEL
LIN {X 0,Y 199.667,Z 396.596,A -85,B 0,C 180,E1 -21558.027,E2 -21558.027} C_VEL
LIN {X 0,Y 199.701,Z 396.608,A -85,B 0,C 180,E1 -21560.734,E2 -21560.734} C_VEL
LIN {X 0,Y 199.631,Z 396.596,A -85,B 0,C 180,E1 -21565.716,E2 -21565.716} C_VEL
LIN {X 0,Y 199.694,Z 396.606,A -85,B 0,C 180,E1 -21568.135,E2 -21568.135} C_VEL
LIN {X 0,Y 199.684,Z 396.598,A -85,B 0,C 180,E1 -21572.771,E2 -21572.771} C_VEL
LIN {X 0,Y 199.747,Z 396.598,A -85,B 0,C 180,E1 -21577.23,E2 -21577.23} C_VEL
LIN {X 0,Y 199.835,Z 396.584,A -85,B 0,C 180,E1 -21581.721,E2 -21581.721} C_VEL
LIN {X 0,Y 199.832,Z 396.574,A -85,B 0,C 180,E1 -21585.747,E2 -21585.747} C_VEL
LIN {X 0,Y 200.067,Z 396.564,A -85,B 0,C 180,E1 -21589.883,E2 -21589.883} C_VEL
LIN {X 0,Y 200.03,Z 396.544,A -85,B 0,C 180,E1 -21593.949,E2 -21593.949} C_VEL
LIN {X 0,Y 200.317,Z 396.523,A -85,B 0,C 180,E1 -21597.989,E2 -21597.989} C_VEL
LIN {X 0,Y 200.478,Z 396.512,A -85,B 0,C 180,E1 -21599.999,E2 -21599.999} C_VEL
LIN {X 0,Y 200.028,Z 396.564,A -85,B 0,C 180,E1 -21604.029,E2 -21604.029} C_VEL
LIN {X 0,Y 200.107,Z 396.554,A -85,B 0,C 180,E1 -21608.075,E2 -21608.075} C_VEL
LIN {X 0,Y 199.909,Z 396.582,A -85,B 0,C 180,E1 -21612.177,E2 -21612.177} C_VEL
LIN {X 0,Y 199.801,Z 396.598,A -85,B 0,C 180,E1 -21616.343,E2 -21616.343} C_VEL
LIN {X 0,Y 199.738,Z 396.605,A -85,B 0,C 180,E1 -21620.601,E2 -21620.601} C_VEL
LIN {X 0,Y 199.672,Z 396.612,A -85,B 0,C 180,E1 -21624.984,E2 -21624.984} C_VEL
LIN {X 0,Y 199.661,Z 396.615,A -85,B 0,C 180,E1 -21629.524,E2 -21629.524} C_VEL
LIN {X 0,Y 199.655,Z 396.617,A -85,B 0,C 180,E1 -21632.35,E2 -21632.35} C_VEL
LIN {X 0,Y 199.65,Z 396.616,A -85,B 0,C 180,E1 -21636.757,E2 -21636.757} C_VEL
LIN {X 0,Y 199.676,Z 396.613,A -85,B 0,C 180,E1 -21639.312,E2 -21639.312} C_VEL
LIN {X 0,Y 199.66,Z 396.612,A -85,B 0,C 180,E1 -21642.338,E2 -21642.338} C_VEL
LIN {X 0,Y 199.644,Z 396.615,A -85,B 0,C 180,E1 -21645.248,E2 -21645.248} C_VEL
LIN {X 0,Y 199.654,Z 396.682,A -85,B 0,C 180,E1 -21648.2,E2 -21648.2} C_VEL
LIN {X 0,Y 201.693,Z 404.926,A -85,B 0,C 180,E1 -21652.496,E2 -21652.496} C_VEL
LIN {X 0,Y 202.011,Z 406.161,A -85,B 0,C 180,E1 -21653.049,E2 -21653.049} C_VEL
LIN {X 0,Y 209.233,Z 422.842,A -85,B 0,C 180,E1 -21654.969,E2 -21654.969} C_VEL
LIN {X 0,Y 209.823,Z 424.281,A -85,B 0,C 180,E1 -21655.122,E2 -21655.122} C_VEL
LIN {X 0,Y 210.949,Z 427.822,A -85,B 0,C 180,E1 -21655.441,E2 -21655.441} C_VEL
LIN {X 0,Y 211.396,Z 431.628,A -85,B 0,C 180,E1 -21655.659,E2 -21655.659} C_VEL
LIN {X 0,Y 210.962,Z 439.521,A -85,B 0,C 180,E1 -21655.896,E2 -21655.896} C_VEL
LIN {X 0,Y 209.51,Z 451.754,A -85,B 0,C 180,E1 -21656.143,E2 -21656.143} C_VEL
LIN {X 0,Y 209.556,Z 455.806,A -85,B 0,C 180,E1 -21656.307,E2 -21656.307} C_VEL
LIN {X 0,Y 210.503,Z 468.484,A -85,B 0,C 180,E1 -21656.94,E2 -21656.94} C_VEL
LIN {X 0,Y 208.483,Z 514.698,A -85,B 0,C 180,E1 -21658.462,E2 -21658.462} C_VEL
LIN {X 0,Y 207.342,Z 527.761,A -85,B 0,C 180,E1 -21659.235,E2 -21659.235} C_VEL
LIN {X 0,Y 205.506,Z 541.124,A -85,B 0,C 180,E1 -21660.414,E2 -21660.414} C_VEL
LIN {X 0,Y 203.374,Z 553.167,A -85,B 0,C 180,E1 -21661.912,E2 -21661.912} C_VEL
LIN {X 0,Y 200.902,Z 564.686,A -85,B 0,C 180,E1 -21663.791,E2 -21663.791} C_VEL
LIN {X 0,Y 198.513,Z 575.08,A -85,B 0,C 180,E1 -21665.976,E2 -21665.976} C_VEL
LIN {X 0,Y 196.215,Z 584.569,A -85,B 0,C 180,E1 -21668.517,E2 -21668.517} C_VEL
LIN {X 0,Y 194.548,Z 592.104,A -85,B 0,C 180,E1 -21671.027,E2 -21671.027} C_VEL
LIN {X 0,Y 192.738,Z 599.627,A -85,B 0,C 180,E1 -21674.129,E2 -21674.129} C_VEL
LIN {X 0,Y 191.406,Z 605.657,A -85,B 0,C 180,E1 -21677.273,E2 -21677.273} C_VEL
LIN {X 0,Y 190.687,Z 610.422,A -85,B 0,C 180,E1 -21680.453,E2 -21680.453} C_VEL
LIN {X 0,Y 190.348,Z 614.046,A -85,B 0,C 180,E1 -21683.641,E2 -21683.641} C_VEL
LIN {X 0,Y 190.315,Z 615.903,A -85,B 0,C 180,E1 -21685.765,E2 -21685.765} C_VEL
LIN {X 0,Y 190.412,Z 617.286,A -85,B 0,C 180,E1 -21687.885,E2 -21687.885} C_VEL
LIN {X 0,Y 190.519,Z 618.26,A -85,B 0,C 180,E1 -21690,E2 -21690} C_VEL
LIN {X 0,Y 190.378,Z 618.821,A -85,B 0,C 180,E1 -21692.116,E2 -21692.116} C_VEL
LIN {X 0,Y 190.244,Z 618.978,A -85,B 0,C 180,E1 -21694.237,E2 -21694.237} C_VEL
LIN {X 0,Y 190.485,Z 618.054,A -85,B 0,C 180,E1 -21698.487,E2 -21698.487} C_VEL
LIN {X 0,Y 191.588,Z 615.59,A -85,B 0,C 180,E1 -21702.714,E2 -21702.714} C_VEL
LIN {X 0,Y 192.994,Z 612.619,A -85,B 0,C 180,E1 -21705.849,E2 -21705.849} C_VEL
LIN {X 0,Y 195.094,Z 608.638,A -85,B 0,C 180,E1 -21708.917,E2 -21708.917} C_VEL
LIN {X 0,Y 197.736,Z 603.545,A -85,B 0,C 180,E1 -21711.912,E2 -21711.912} C_VEL
LIN {X 0,Y 200.664,Z 597.171,A -85,B 0,C 180,E1 -21714.852,E2 -21714.852} C_VEL
LIN {X 0,Y 204.306,Z 589.232,A -85,B 0,C 180,E1 -21717.67,E2 -21717.67} C_VEL
LIN {X 0,Y 207.868,Z 581.169,A -85,B 0,C 180,E1 -21719.913,E2 -21719.913} C_VEL
LIN {X 0,Y 211.706,Z 571.358,A -85,B 0,C 180,E1 -21722.082,E2 -21722.082} C_VEL
LIN {X 0,Y 215.472,Z 560.415,A -85,B 0,C 180,E1 -21723.956,E2 -21723.956} C_VEL
LIN {X 0,Y 219.006,Z 547.955,A -85,B 0,C 180,E1 -21725.565,E2 -21725.565} C_VEL
LIN {X 0,Y 221.872,Z 535.706,A -85,B 0,C 180,E1 -21726.717,E2 -21726.717} C_VEL
LIN {X 0,Y 224.035,Z 522.811,A -85,B 0,C 180,E1 -21727.569,E2 -21727.569} C_VEL
LIN {X 0,Y 225.443,Z 509.172,A -85,B 0,C 180,E1 -21728.14,E2 -21728.14} C_VEL
LIN {X 0,Y 227.447,Z 472.161,A -85,B 0,C 180,E1 -21729.248,E2 -21729.248} C_VEL
LIN {X 0,Y 225.967,Z 460.702,A -85,B 0,C 180,E1 -21730.091,E2 -21730.091} C_VEL
LIN {X 0,Y 220.005,Z 446.828,A -85,B 0,C 180,E1 -21732.23,E2 -21732.23} C_VEL
LIN {X 0,Y 213.766,Z 434.416,A -85,B 0,C 180,E1 -21734.593,E2 -21734.593} C_VEL
LIN {X 0,Y 208.206,Z 424.666,A -85,B 0,C 180,E1 -21736.859,E2 -21736.859} C_VEL
LIN {X 0,Y 204.843,Z 419.159,A -85,B 0,C 180,E1 -21738.324,E2 -21738.324} C_VEL
LIN {X 0,Y 202.018,Z 414.636,A -85,B 0,C 180,E1 -21739.628,E2 -21739.628} C_VEL
LIN {X 0,Y 198.905,Z 409.666,A -85,B 0,C 180,E1 -21741.158,E2 -21741.158} C_VEL
LIN {X 0,Y 195.238,Z 404.872,A -85,B 0,C 180,E1 -21743.038,E2 -21743.038} C_VEL
LIN {X 0,Y 194.347,Z 403.075,A -85,B 0,C 180,E1 -21743.639,E2 -21743.639} C_VEL
LIN {X 0,Y 192.613,Z 397.488,A -85,B 0,C 180,E1 -21748.824,E2 -21748.824} C_VEL
LIN {X 0,Y 192.661,Z 397.487,A -85,B 0,C 180,E1 -21751.692,E2 -21751.692} C_VEL
LIN {X 0,Y 192.702,Z 397.448,A -85,B 0,C 180,E1 -21756.349,E2 -21756.349} C_VEL
LIN {X 0,Y 192.728,Z 397.468,A -85,B 0,C 180,E1 -21761.458,E2 -21761.458} C_VEL
LIN {X 0,Y 192.848,Z 397.464,A -85,B 0,C 180,E1 -21767.37,E2 -21767.37} C_VEL
LIN {X 0,Y 193.064,Z 397.437,A -85,B 0,C 180,E1 -21771.628,E2 -21771.628} C_VEL
LIN {X 0,Y 193.26,Z 397.402,A -85,B 0,C 180,E1 -21777.916,E2 -21777.916} C_VEL
LIN {X 0,Y 193.442,Z 397.381,A -85,B 0,C 180,E1 -21780.001,E2 -21780.001} C_VEL
LIN {X 0,Y 192.969,Z 397.436,A -85,B 0,C 180,E1 -21784.178,E2 -21784.178} C_VEL
LIN {X 0,Y 193.033,Z 397.428,A -85,B 0,C 180,E1 -21788.375,E2 -21788.375} C_VEL
LIN {X 0,Y 192.797,Z 397.458,A -85,B 0,C 180,E1 -21792.634,E2 -21792.634} C_VEL
LIN {X 0,Y 192.766,Z 397.463,A -85,B 0,C 180,E1 -21796.959,E2 -21796.959} C_VEL
LIN {X 0,Y 192.639,Z 397.48,A -85,B 0,C 180,E1 -21801.398,E2 -21801.398} C_VEL
LIN {X 0,Y 192.662,Z 397.468,A -85,B 0,C 180,E1 -21804.225,E2 -21804.225} C_VEL
LIN {X 0,Y 192.618,Z 397.457,A -85,B 0,C 180,E1 -21806.915,E2 -21806.915} C_VEL
LIN {X 0,Y 193.584,Z 400.211,A -85,B 0,C 180,E1 -21807.574,E2 -21807.574} C_VEL
LIN {X 0,Y 195.728,Z 402.485,A -85,B 0,C 180,E1 -21808.712,E2 -21808.712} C_VEL
LIN {X 0,Y 196.765,Z 403.286,A -85,B 0,C 180,E1 -21809.222,E2 -21809.222} C_VEL
LIN {X 0,Y 198.842,Z 406.651,A -85,B 0,C 180,E1 -21810.317,E2 -21810.317} C_VEL
LIN {X 0,Y 200.679,Z 408.517,A -85,B 0,C 180,E1 -21811.176,E2 -21811.176} C_VEL
LIN {X 0,Y 203.299,Z 412.172,A -85,B 0,C 180,E1 -21812.401,E2 -21812.401} C_VEL
LIN {X 0,Y 205.054,Z 414.583,A -85,B 0,C 180,E1 -21813.184,E2 -21813.184} C_VEL
LIN {X 0,Y 208.182,Z 418.826,A -85,B 0,C 180,E1 -21814.508,E2 -21814.508} C_VEL
LIN {X 0,Y 212.898,Z 425.509,A -85,B 0,C 180,E1 -21816.383,E2 -21816.383} C_VEL
LIN {X 0,Y 219.559,Z 436.189,A -85,B 0,C 180,E1 -21818.844,E2 -21818.844} C_VEL
LIN {X 0,Y 224.707,Z 445.326,A -85,B 0,C 180,E1 -21820.613,E2 -21820.613} C_VEL
LIN {X 0,Y 228.42,Z 453.461,A -85,B 0,C 180,E1 -21821.874,E2 -21821.874} C_VEL
LIN {X 0,Y 225.82,Z 498.622,A -85,B 0,C 180,E1 -21823.25,E2 -21823.25} C_VEL
LIN {X 0,Y 224.355,Z 511.069,A -85,B 0,C 180,E1 -21823.907,E2 -21823.907} C_VEL
LIN {X 0,Y 222.24,Z 524.081,A -85,B 0,C 180,E1 -21824.963,E2 -21824.963} C_VEL
LIN {X 0,Y 219.489,Z 535.486,A -85,B 0,C 180,E1 -21826.179,E2 -21826.179} C_VEL
LIN {X 0,Y 216.481,Z 546.198,A -85,B 0,C 180,E1 -21827.715,E2 -21827.715} C_VEL
LIN {X 0,Y 213.144,Z 556.75,A -85,B 0,C 180,E1 -21829.689,E2 -21829.689} C_VEL
LIN {X 0,Y 209.809,Z 565.458,A -85,B 0,C 180,E1 -21831.707,E2 -21831.707} C_VEL
LIN {X 0,Y 206.408,Z 573.474,A -85,B 0,C 180,E1 -21834.032,E2 -21834.032} C_VEL
LIN {X 0,Y 202.749,Z 581.248,A -85,B 0,C 180,E1 -21836.911,E2 -21836.911} C_VEL
LIN {X 0,Y 200.037,Z 586.529,A -85,B 0,C 180,E1 -21839.375,E2 -21839.375} C_VEL
LIN {X 0,Y 197.254,Z 591.602,A -85,B 0,C 180,E1 -21842.408,E2 -21842.408} C_VEL
LIN {X 0,Y 194.909,Z 595.505,A -85,B 0,C 180,E1 -21845.502,E2 -21845.502} C_VEL
LIN {X 0,Y 193.112,Z 598.344,A -85,B 0,C 180,E1 -21848.659,E2 -21848.659} C_VEL
LIN {X 0,Y 191.619,Z 600.426,A -85,B 0,C 180,E1 -21852.481,E2 -21852.481} C_VEL
LIN {X 0,Y 190.926,Z 601.114,A -85,B 0,C 180,E1 -21855.068,E2 -21855.068} C_VEL
LIN {X 0,Y 190.47,Z 601.205,A -85,B 0,C 180,E1 -21857.21,E2 -21857.21} C_VEL
LIN {X 0,Y 190.263,Z 600.199,A -85,B 0,C 180,E1 -21861.503,E2 -21861.503} C_VEL
LIN {X 0,Y 190.552,Z 598.334,A -85,B 0,C 180,E1 -21864.772,E2 -21864.772} C_VEL
LIN {X 0,Y 191.029,Z 594.511,A -85,B 0,C 180,E1 -21868.946,E2 -21868.946} C_VEL
LIN {X 0,Y 191.918,Z 590.394,A -85,B 0,C 180,E1 -21872.099,E2 -21872.099} C_VEL
LIN {X 0,Y 193.324,Z 584.121,A -85,B 0,C 180,E1 -21875.737,E2 -21875.737} C_VEL
LIN {X 0,Y 195.1,Z 577.287,A -85,B 0,C 180,E1 -21878.806,E2 -21878.806} C_VEL
LIN {X 0,Y 197.299,Z 568.746,A -85,B 0,C 180,E1 -21881.819,E2 -21881.819} C_VEL
LIN {X 0,Y 199.442,Z 559.987,A -85,B 0,C 180,E1 -21884.28,E2 -21884.28} C_VEL
LIN {X 0,Y 201.702,Z 550.364,A -85,B 0,C 180,E1 -21886.445,E2 -21886.445} C_VEL
LIN {X 0,Y 203.869,Z 539.845,A -85,B 0,C 180,E1 -21888.334,E2 -21888.334} C_VEL
LIN {X 0,Y 205.738,Z 528.195,A -85,B 0,C 180,E1 -21889.974,E2 -21889.974} C_VEL
LIN {X 0,Y 207.395,Z 516.067,A -85,B 0,C 180,E1 -21891.233,E2 -21891.233} C_VEL
LIN {X 0,Y 208.633,Z 502.661,A -85,B 0,C 180,E1 -21892.217,E2 -21892.217} C_VEL
LIN {X 0,Y 209.364,Z 489.262,A -85,B 0,C 180,E1 -21892.791,E2 -21892.791} C_VEL
LIN {X 0,Y 211.526,Z 435.946,A -85,B 0,C 180,E1 -21894.512,E2 -21894.512} C_VEL
LIN {X 0,Y 208.48,Z 428.073,A -85,B 0,C 180,E1 -21895.305,E2 -21895.305} C_VEL
LIN {X 0,Y 200.076,Z 411.17,A -85,B 0,C 180,E1 -21897.455,E2 -21897.455} C_VEL
LIN {X 0,Y 194.183,Z 401.09,A -85,B 0,C 180,E1 -21899.027,E2 -21899.027} C_VEL
LIN {X 0,Y 192.886,Z 398.589,A -85,B 0,C 180,E1 -21899.402,E2 -21899.402} C_VEL
LIN {X 0,Y 192.653,Z 397.485,A -85,B 0,C 180,E1 -21899.573,E2 -21899.573} C_VEL
LIN {X 0,Y 192.601,Z 397.494,A -85,B 0,C 180,E1 -21903.184,E2 -21903.184} C_VEL
LIN {X 0,Y 192.553,Z 397.5,A -85,B 0,C 180,E1 -21908.35,E2 -21908.35} C_VEL
LIN {X 0,Y 192.537,Z 397.499,A -85,B 0,C 180,E1 -21913.109,E2 -21913.109} C_VEL
LIN {X 0,Y 192.6,Z 397.476,A -85,B 0,C 180,E1 -21916.868,E2 -21916.868} C_VEL
LIN {X 0,Y 192.612,Z 397.491,A -85,B 0,C 180,E1 -21921.661,E2 -21921.661} C_VEL
LIN {X 0,Y 192.596,Z 397.48,A -85,B 0,C 180,E1 -21926.813,E2 -21926.813} C_VEL
LIN {X 0,Y 192.659,Z 397.48,A -85,B 0,C 180,E1 -21931.69,E2 -21931.69} C_VEL
LIN {X 0,Y 192.709,Z 397.467,A -85,B 0,C 180,E1 -21936.348,E2 -21936.348} C_VEL
LIN {X 0,Y 192.779,Z 397.466,A -85,B 0,C 180,E1 -21941.412,E2 -21941.412} C_VEL
LIN {X 0,Y 192.76,Z 397.45,A -85,B 0,C 180,E1 -21945.213,E2 -21945.213} C_VEL
LIN {X 0,Y 192.978,Z 397.445,A -85,B 0,C 180,E1 -21949.508,E2 -21949.508} C_VEL
LIN {X 0,Y 193.058,Z 397.431,A -85,B 0,C 180,E1 -21951.627,E2 -21951.627} C_VEL
LIN {X 0,Y 193.259,Z 397.402,A -85,B 0,C 180,E1 -21957.915,E2 -21957.915} C_VEL
LIN {X 0,Y 193.442,Z 397.388,A -85,B 0,C 180,E1 -21959.999,E2 -21959.999} C_VEL
LIN {X 0,Y 192.974,Z 397.443,A -85,B 0,C 180,E1 -21964.177,E2 -21964.177} C_VEL
LIN {X 0,Y 193.058,Z 397.431,A -85,B 0,C 180,E1 -21968.372,E2 -21968.372} C_VEL
LIN {X 0,Y 192.848,Z 397.459,A -85,B 0,C 180,E1 -21972.63,E2 -21972.63} C_VEL
LIN {X 0,Y 192.778,Z 397.465,A -85,B 0,C 180,E1 -21978.587,E2 -21978.587} C_VEL
LIN {X 0,Y 192.665,Z 397.483,A -85,B 0,C 180,E1 -21984.227,E2 -21984.227} C_VEL
LIN {X 0,Y 192.641,Z 397.488,A -85,B 0,C 180,E1 -21988.889,E2 -21988.889} C_VEL
LIN {X 0,Y 192.595,Z 397.496,A -85,B 0,C 180,E1 -21993.186,E2 -21993.186} C_VEL
LIN {X 0,Y 192.598,Z 397.495,A -85,B 0,C 180,E1 -21998.341,E2 -21998.341} C_VEL
LIN {X 0,Y 192.599,Z 397.494,A -85,B 0,C 180,E1 -22003.131,E2 -22003.131} C_VEL
LIN {X 0,Y 192.568,Z 397.564,A -85,B 0,C 180,E1 -22007.2,E2 -22007.2} C_VEL
LIN {X 0,Y 194.66,Z 405.698,A -85,B 0,C 180,E1 -22011.63,E2 -22011.63} C_VEL
LIN {X 0,Y 202.305,Z 422.739,A -85,B 0,C 180,E1 -22013.788,E2 -22013.788} C_VEL
LIN {X 0,Y 207.463,Z 436.333,A -85,B 0,C 180,E1 -22015.212,E2 -22015.212} C_VEL
LIN {X 0,Y 209.556,Z 455.806,A -85,B 0,C 180,E1 -22016.307,E2 -22016.307} C_VEL
LIN {X 0,Y 209.532,Z 459.705,A -85,B 0,C 180,E1 -22016.454,E2 -22016.454} C_VEL
LIN {X 0,Y 208.578,Z 465.552,A -85,B 0,C 180,E1 -22016.534,E2 -22016.534} C_VEL
LIN {X 0,Y 204.773,Z 479.044,A -85,B 0,C 180,E1 -22016.471,E2 -22016.471} C_VEL
LIN {X 0,Y 203.672,Z 484.931,A -85,B 0,C 180,E1 -22016.531,E2 -22016.531} C_VEL
LIN {X 0,Y 203.519,Z 486.913,A -85,B 0,C 180,E1 -22016.586,E2 -22016.586} C_VEL
LIN {X 0,Y 202.118,Z 515.616,A -85,B 0,C 180,E1 -22017.589,E2 -22017.589} C_VEL
LIN {X 0,Y 200.885,Z 528.769,A -85,B 0,C 180,E1 -22018.421,E2 -22018.421} C_VEL
LIN {X 0,Y 198.991,Z 541.747,A -85,B 0,C 180,E1 -22019.637,E2 -22019.637} C_VEL
LIN {X 0,Y 196.776,Z 553.564,A -85,B 0,C 180,E1 -22021.174,E2 -22021.174} C_VEL
LIN {X 0,Y 194.221,Z 564.95,A -85,B 0,C 180,E1 -22023.108,E2 -22023.108} C_VEL
LIN {X 0,Y 191.748,Z 575.213,A -85,B 0,C 180,E1 -22025.36,E2 -22025.36} C_VEL
LIN {X 0,Y 189.163,Z 585.267,A -85,B 0,C 180,E1 -22028.19,E2 -22028.19} C_VEL
LIN {X 0,Y 187.411,Z 592.768,A -85,B 0,C 180,E1 -22030.845,E2 -22030.845} C_VEL
LIN {X 0,Y 185.594,Z 600.117,A -85,B 0,C 180,E1 -22034.066,E2 -22034.066} C_VEL
LIN {X 0,Y 184.423,Z 605.073,A -85,B 0,C 180,E1 -22036.783,E2 -22036.783} C_VEL
LIN {X 0,Y 183.665,Z 609.893,A -85,B 0,C 180,E1 -22040.085,E2 -22040.085} C_VEL
LIN {X 0,Y 183.286,Z 613.568,A -85,B 0,C 180,E1 -22043.395,E2 -22043.395} C_VEL
LIN {X 0,Y 183.233,Z 615.563,A -85,B 0,C 180,E1 -22045.74,E2 -22045.74} C_VEL
LIN {X 0,Y 183.309,Z 616.875,A -85,B 0,C 180,E1 -22047.803,E2 -22047.803} C_VEL
LIN {X 0,Y 183.433,Z 617.872,A -85,B 0,C 180,E1 -22050,E2 -22050} C_VEL
LIN {X 0,Y 183.292,Z 618.454,A -85,B 0,C 180,E1 -22052.197,E2 -22052.197} C_VEL
LIN {X 0,Y 183.154,Z 618.642,A -85,B 0,C 180,E1 -22054.401,E2 -22054.401} C_VEL
LIN {X 0,Y 183.203,Z 618.405,A -85,B 0,C 180,E1 -22056.608,E2 -22056.608} C_VEL
LIN {X 0,Y 183.934,Z 616.759,A -85,B 0,C 180,E1 -22061.014,E2 -22061.014} C_VEL
LIN {X 0,Y 184.63,Z 615.357,A -85,B 0,C 180,E1 -22063.202,E2 -22063.202} C_VEL
LIN {X 0,Y 186.152,Z 612.428,A -85,B 0,C 180,E1 -22066.448,E2 -22066.448} C_VEL
LIN {X 0,Y 188.352,Z 608.495,A -85,B 0,C 180,E1 -22069.622,E2 -22069.622} C_VEL
LIN {X 0,Y 191.13,Z 603.455,A -85,B 0,C 180,E1 -22072.711,E2 -22072.711} C_VEL
LIN {X 0,Y 194.217,Z 597.153,A -85,B 0,C 180,E1 -22075.736,E2 -22075.736} C_VEL
LIN {X 0,Y 198.054,Z 589.299,A -85,B 0,C 180,E1 -22078.623,E2 -22078.623} C_VEL
LIN {X 0,Y 202.521,Z 579.538,A -85,B 0,C 180,E1 -22081.367,E2 -22081.367} C_VEL
LIN {X 0,Y 206.594,Z 569.434,A -85,B 0,C 180,E1 -22083.558,E2 -22083.558} C_VEL
LIN {X 0,Y 210.538,Z 558.019,A -85,B 0,C 180,E1 -22085.449,E2 -22085.449} C_VEL
LIN {X 0,Y 213.803,Z 546.827,A -85,B 0,C 180,E1 -22086.862,E2 -22086.862} C_VEL
LIN {X 0,Y 216.76,Z 534.258,A -85,B 0,C 180,E1 -22088.026,E2 -22088.026} C_VEL
LIN {X 0,Y 218.975,Z 520.702,A -85,B 0,C 180,E1 -22088.903,E2 -22088.903} C_VEL
LIN {X 0,Y 220.313,Z 507.233,A -85,B 0,C 180,E1 -22089.435,E2 -22089.435} C_VEL
LIN {X 0,Y 222.189,Z 472.676,A -85,B 0,C 180,E1 -22090.497,E2 -22090.497} C_VEL
LIN {X 0,Y 221.021,Z 463.66,A -85,B 0,C 180,E1 -22091.196,E2 -22091.196} C_VEL
LIN {X 0,Y 215.782,Z 451.254,A -85,B 0,C 180,E1 -22093.185,E2 -22093.185} C_VEL
LIN {X 0,Y 209.73,Z 438.937,A -85,B 0,C 180,E1 -22095.612,E2 -22095.612} C_VEL
LIN {X 0,Y 204.635,Z 429.797,A -85,B 0,C 180,E1 -22097.805,E2 -22097.805} C_VEL
LIN {X 0,Y 200.803,Z 423.371,A -85,B 0,C 180,E1 -22099.579,E2 -22099.579} C_VEL
LIN {X 0,Y 198.683,Z 419.913,A -85,B 0,C 180,E1 -22100.619,E2 -22100.619} C_VEL
LIN {X 0,Y 195.215,Z 414.538,A -85,B 0,C 180,E1 -22102.415,E2 -22102.415} C_VEL
LIN {X 0,Y 191.961,Z 409.794,A -85,B 0,C 180,E1 -22104.223,E2 -22104.223} C_VEL
LIN {X 0,Y 190.029,Z 407.372,A -85,B 0,C 180,E1 -22105.346,E2 -22105.346} C_VEL
LIN {X 0,Y 187.012,Z 402.873,A -85,B 0,C 180,E1 -22107.284,E2 -22107.284} C_VEL
LIN {X 0,Y 186.741,Z 402.144,A -85,B 0,C 180,E1 -22107.748,E2 -22107.748} C_VEL
LIN {X 0,Y 185.632,Z 398.36,A -85,B 0,C 180,E1 -22111.755,E2 -22111.755} C_VEL
LIN {X 0,Y 185.583,Z 398.328,A -85,B 0,C 180,E1 -22115.382,E2 -22115.382} C_VEL
LIN {X 0,Y 185.604,Z 398.356,A -85,B 0,C 180,E1 -22120.075,E2 -22120.075} C_VEL
LIN {X 0,Y 185.695,Z 398.343,A -85,B 0,C 180,E1 -22124.638,E2 -22124.638} C_VEL
LIN {X 0,Y 185.921,Z 398.313,A -85,B 0,C 180,E1 -22129.359,E2 -22129.359} C_VEL
LIN {X 0,Y 185.961,Z 398.309,A -85,B 0,C 180,E1 -22133.49,E2 -22133.49} C_VEL
LIN {X 0,Y 186.204,Z 398.281,A -85,B 0,C 180,E1 -22137.837,E2 -22137.837} C_VEL
LIN {X 0,Y 186.405,Z 398.258,A -85,B 0,C 180,E1 -22140.001,E2 -22140.001} C_VEL
LIN {X 0,Y 185.916,Z 398.315,A -85,B 0,C 180,E1 -22144.337,E2 -22144.337} C_VEL
LIN {X 0,Y 185.979,Z 398.307,A -85,B 0,C 180,E1 -22148.695,E2 -22148.695} C_VEL
LIN {X 0,Y 185.725,Z 398.339,A -85,B 0,C 180,E1 -22153.124,E2 -22153.124} C_VEL
LIN {X 0,Y 185.713,Z 398.342,A -85,B 0,C 180,E1 -22157.623,E2 -22157.623} C_VEL
LIN {X 0,Y 185.646,Z 398.505,A -85,B 0,C 180,E1 -22163.275,E2 -22163.275} C_VEL
LIN {X 0,Y 186.66,Z 401.248,A -85,B 0,C 180,E1 -22164.08,E2 -22164.08} C_VEL
LIN {X 0,Y 188.703,Z 403.38,A -85,B 0,C 180,E1 -22165.361,E2 -22165.361} C_VEL
LIN {X 0,Y 190.035,Z 404.354,A -85,B 0,C 180,E1 -22166.125,E2 -22166.125} C_VEL
LIN {X 0,Y 191.866,Z 407.373,A -85,B 0,C 180,E1 -22167.251,E2 -22167.251} C_VEL
LIN {X 0,Y 194.185,Z 409.734,A -85,B 0,C 180,E1 -22168.497,E2 -22168.497} C_VEL
LIN {X 0,Y 196.641,Z 413.202,A -85,B 0,C 180,E1 -22169.803,E2 -22169.803} C_VEL
LIN {X 0,Y 198.129,Z 414.976,A -85,B 0,C 180,E1 -22170.539,E2 -22170.539} C_VEL
LIN {X 0,Y 201.877,Z 420.188,A -85,B 0,C 180,E1 -22172.331,E2 -22172.331} C_VEL
LIN {X 0,Y 207.159,Z 427.508,A -85,B 0,C 180,E1 -22174.629,E2 -22174.629} C_VEL
LIN {X 0,Y 213.873,Z 438.101,A -85,B 0,C 180,E1 -22177.309,E2 -22177.309} C_VEL
